// TwinCAT 3 PLC project BX130XPLC
// ProgramVersion: 3.1.4024.0
// libraries:
//   Tc2_EtherCAT, * (Beckhoff Automation GmbH)
//   Tc2_MC2, * (Beckhoff Automation GmbH)
//   Tc2_ModbusSrv, * (Beckhoff Automation GmbH)
//   Tc2_NcDrive, * (Beckhoff Automation GmbH)
//   Tc2_Standard, * (Beckhoff Automation GmbH)
//   Tc2_System, * (Beckhoff Automation GmbH)
//   Tc2_Utilities, * (Beckhoff Automation GmbH)
//   Tc3_Module, * (Beckhoff Automation GmbH)
//   TcMatrix, * (Burks Engineering)
// project tree:
//   DUTs/ E_MachineState.TcTLEO, E_ProgramMap.TcDUT, Program_Type.TcDUT, Structure_Error.TcDUT, Structure_RobotPose.TcDUT, Tool_Type.TcDUT
//   GVLs/ GVL_Axes.TcGVL, GVL_OperationCounter.TcGVL, GVL_Programs.TcGVL, GVL_SERVO_ROBOT_CONST.TcGVL
//   / PlcTask.TcTTO
//   POUs/Components/ FB_Enclosure.TcPOU, FB_GantryHoldDown.TcPOU, FB_OperatingCounter.TcPOU, FB_Robot.TcPOU, FB_Spindle.TcPOU, FB_TorqueSensor.TcPOU
//   POUs/ FB_Machine.TcPOU, MAIN.TcPOU
// real-time tasks:
//   TASK PlcTask: cycle T#10ms, priority 20, ADS port 350
// motion (NC):
//   TASK NC-Task 1 SAF: cycle T#2ms, priority 4, ADS port 501
//   TASK NC-Task 1 SVB: cycle T#10ms, priority 8, ADS port 511
//   AXIS Axis West (id 1)
//     Dynamic: Acceleration=260.052, Deceleration=260.052, Jerk=780.156
//     Velo: RefSync=10, SlowManual=8.6684051275234, FastManual=52.0104307651404, Fast=173.368102550468, Maximum=173.368
//     OtherSettings: AllowMotionCmdToSlave=true
//     encoder EncType=8
//       EncPara: ScaleFactorNumerator=9.999689, ScaleFactorDenominator=1048576, Inverse=true, MaxCount=#xffffffff
//         SoftEndMinControl: Enable=true, Range=1
//         SoftEndMaxControl: Enable=true, Range=2335
//         Inc: RefSearchInverse=true, RefSyncInverse=false
//     drive DrvType=9
//       DrvPara: Inverse=true, MaxCount=#xffffffff, DriveControlDWord=#x00030100
//         Analog: VeloReferenz=190.704912805515, VeloScale=1.02400649589962, TorqueSetpointScale=10, ScaleFactorActTorque=0.1
//         TimeComp: TaskDelayCycles=1
//     controller CtrType=1
//       CtrPara: PriorControlFactor=1
//         Observer: BandWidth=20
//   AXIS Axis East (id 2)
//     Dynamic: Acceleration=260.052, Deceleration=260.052, Jerk=780.156
//     Velo: RefSearch=1.73368102550468, RefSync=1.73368102550468, SlowManual=8.6684051275234, FastManual=52.0104307651404, Fast=173.368102550468, Maximum=173.368
//     OtherSettings: AllowMotionCmdToSlave=true
//     encoder EncType=8
//       EncPara: ScaleFactorNumerator=9.999689, ScaleFactorDenominator=1048576, MaxCount=#xffffffff
//         SoftEndMaxControl: Range=2377
//         Inc: RefSearchInverse=true, RefSyncInverse=false
//     drive DrvType=9
//       DrvPara: MaxCount=#xffffffff, DriveControlDWord=#x00030100
//         Analog: VeloReferenz=190.704912805515, VeloScale=1.02400649589962, TorqueSetpointScale=10, ScaleFactorActTorque=0.1
//         TimeComp: TaskDelayCycles=1
//     controller CtrType=1
//       CtrPara: PriorControlFactor=1
//         Observer: BandWidth=20
// I/O:
//   DEVICE PortLAN1X102, AmsNetId 172.18.239.23.3.1
//     Term 1 (EK1100) [EK1100 EtherCAT Coupler (2A E-Bus)]
//       Term 2 (EL1918) [EL1918, 8Ch. Safety Input 24V, TwinSAFE]
//         modules: Module 1 (FSOE), Module 2 (FSLOGIC)
//       Term 3 (EL1918) [EL1918, 8Ch. Safety Input 24V, TwinSAFE]
//         modules: Module 2 (FSLOGIC)
//       Term 4 (EL2904) [EL2904, 4 Ch. Safety Output 24V, 0.5A, TwinSAFE]
//         modules: Module 1 (FSOES), Module 2 (DO)
//       Term 5 (EL1008) [EL1008 8Ch. Dig. Input 24V, 3ms]
//       Term 6 (EL1008) [EL1008 8Ch. Dig. Input 24V, 3ms]
//       Term 7 (EL1008) [EL1008 8Ch. Dig. Input 24V, 3ms]
//       Term 8 (EL9410) [EL9410 E-Bus Power Supplier  (Diagnostics)]
//       Term 9 (EL2008) [EL2008 8Ch. Dig. Output 24V, 0.5A]
//       Term 10 (EL2008) [EL2008 8Ch. Dig. Output 24V, 0.5A]
//       Term 11 (EL2008) [EL2008 8Ch. Dig. Output 24V, 0.5A]
//       Term 27 (EL1008) [EL1008 8Ch. Dig. Input 24V, 3ms]
//       Term 12 (EK1122) [EK1122 2 port EtherCAT junction]
//         Term 30 (ATI Axia F/T Sensor) [ATI Axia F/T Sensor]
//       Term 15 (EL9011) [EL9011 End Terminal]
//     Drive 13 (AX5206-0000-0214) [AX5206-0000-0214 EtherCAT Drive (SoE, 2 Ch.)]
//     Box 14 (ECT I/F for KHI Robot Controller) [ECT I/F for KHI Robot Controller]
// variable links:
//   PortLAN1X102 <-> PortLAN1X102/Term 1 (EK1100)/Term 3 (EL1918)
//     Term 1 (EK1100)/Term 2 (EL1918)/Module 1 (FSOE)/FSoE Inputs/FSOE <-> ConnectionOutputs/Message_3 RxPDO
//     Term 1 (EK1100)/Term 2 (EL1918)/Module 1 (FSOE)/FSoE Outputs/FSOE <-> ConnectionInputs/Message_3 TxPDO
//     Term 1 (EK1100)/Term 4 (EL2904)/Module 1 (FSOES)/TxPDO/FSOE <-> ConnectionOutputs/Message_4 RxPDO
//   PortLAN1X102 <-> PortLAN1X102/Term 1 (EK1100)/Term 4 (EL2904)
//     Term 1 (EK1100)/Term 3 (EL1918)/ConnectionInputs/Message_4 TxPDO <-> Module 1 (FSOES)/RxPDO/FSOE
//   NC-Task 1 SAF/Axes/Axis East <-> PortLAN1X102/Drive 13 (AX5206-0000-0214)
//     Drive/Inputs/In/nDataIn1 <-> AT 2/Following distance
//     Drive/Inputs/In/nDataIn3[0] <-> AT 2/Torque/force feedback value
//     Drive/Inputs/In/nDcOutputTime <-> InfoData/DcOutputShift
//     Drive/Inputs/In/nState1 <-> AT 2/Drive status word @bit 8
//     Drive/Inputs/In/nState2 <-> AT 2/Drive status word
//     Drive/Inputs/In/nState4 @bit 1 <-> WcState/InputToggle
//     Drive/Inputs/In/nState4 <-> WcState/WcState
//     Drive/Outputs/Out/nCtrl1 <-> MDT 2/Master control word @bit 8
//     Drive/Outputs/Out/nDataOut1 <-> MDT 2/Position command value
//     Enc/Inputs/In/nDataIn1 <-> AT 2/Position feedback 1 value (motor feedback)
//     Enc/Inputs/In/nDcInputTime <-> InfoData/DcInputShift
//     Enc/Inputs/In/nState4 @bit 1 <-> WcState/InputToggle
//     Enc/Inputs/In/nState4 <-> WcState/WcState
//   NC-Task 1 SAF/Axes/Axis West <-> PortLAN1X102/Drive 13 (AX5206-0000-0214)
//     Drive/Inputs/In/nDataIn1 <-> AT 1/Following distance
//     Drive/Inputs/In/nDataIn3[0] <-> AT 1/Torque/force feedback value
//     Drive/Inputs/In/nDcOutputTime <-> InfoData/DcOutputShift
//     Drive/Inputs/In/nState1 <-> AT 1/Drive status word @bit 8
//     Drive/Inputs/In/nState2 <-> AT 1/Drive status word
//     Drive/Inputs/In/nState4 @bit 1 <-> WcState/InputToggle
//     Drive/Inputs/In/nState4 <-> WcState/WcState
//     Drive/Outputs/Out/nCtrl1 <-> MDT 1/Master control word @bit 8
//     Drive/Outputs/Out/nDataOut1 <-> MDT 1/Position command value
//     Enc/Inputs/In/nDataIn1 <-> AT 1/Position feedback 1 value (motor feedback)
//     Enc/Inputs/In/nDcInputTime <-> InfoData/DcInputShift
//     Enc/Inputs/In/nState4 @bit 1 <-> WcState/InputToggle
//     Enc/Inputs/In/nState4 <-> WcState/WcState
//   BX130XPLC/BX130XPLC Instance <-> PortLAN1X102/Box 14 (ECT I/F for KHI Robot Controller)
//     PlcTask Inputs/MAIN.fbMachine.fbRobot.jt1_pose_1 <-> TxPDO/1-8
//     PlcTask Inputs/MAIN.fbMachine.fbRobot.jt1_pose_2 <-> TxPDO/9-16
//     PlcTask Inputs/MAIN.fbMachine.fbRobot.jt2_pose_1 <-> TxPDO/17-24
//     PlcTask Inputs/MAIN.fbMachine.fbRobot.jt2_pose_2 <-> TxPDO/25-32
//     PlcTask Inputs/MAIN.fbMachine.fbRobot.jt3_pose_1 <-> TxPDO/33-40
//     PlcTask Inputs/MAIN.fbMachine.fbRobot.jt3_pose_2 <-> TxPDO/41-48
//     PlcTask Inputs/MAIN.fbMachine.fbRobot.jt4_pose_1 <-> TxPDO/49-56
//     PlcTask Inputs/MAIN.fbMachine.fbRobot.jt4_pose_2 <-> TxPDO/57-64
//     PlcTask Inputs/MAIN.fbMachine.fbRobot.jt5_pose_1 <-> TxPDO/65-72
//     PlcTask Inputs/MAIN.fbMachine.fbRobot.jt5_pose_2 <-> TxPDO/73-80
//     PlcTask Inputs/MAIN.fbMachine.fbRobot.jt6_pose_1 <-> TxPDO/81-88
//     PlcTask Inputs/MAIN.fbMachine.fbRobot.jt6_pose_2 <-> TxPDO/89-96
//     PlcTask Inputs/MAIN.fbMachine.fbRobot.sigs105112 <-> TxPDO/105-112
//     PlcTask Inputs/MAIN.fbMachine.fbRobot.sigs113120 <-> TxPDO/113-120
//     PlcTask Inputs/MAIN.fbMachine.fbRobot.sigs145152 <-> TxPDO/145-152
//     PlcTask Inputs/MAIN.fbMachine.fbRobot.sigs153160 <-> TxPDO/153-160
//     PlcTask Inputs/MAIN.fbMachine.fbRobot.sigs161168 <-> TxPDO/161-168
//     PlcTask Inputs/MAIN.fbMachine.fbRobot.sigs169176 <-> TxPDO/169-176
//     PlcTask Inputs/MAIN.fbMachine.fbRobot.sigs177184 <-> TxPDO/177-184
//     PlcTask Inputs/MAIN.fbMachine.fbRobot.sigs97104 <-> TxPDO/97-104
//     PlcTask Inputs/MAIN.fbMachine.fbRobot.ztool_pose_1 <-> TxPDO/129-136
//     PlcTask Inputs/MAIN.fbMachine.fbRobot.ztool_pose_2 <-> TxPDO/137-144
//     PlcTask Outputs/MAIN.fbMachine.fbRobot.sigs{10011008..10411048 step 80008} <-> RxPDO/{1001..1041 step 8}-{1008..1048 step 8}  (6 links)
//   BX130XPLC/BX130XPLC Instance <-> PortLAN1X102/Term 1 (EK1100)/Term 10 (EL2008)
//     PlcTask Outputs/MAIN.fbMachine.fbEnclosure.enableRollingDoor <-> Channel 3/enableRollingDoor
//     PlcTask Outputs/MAIN.fbMachine.fbEnclosure.openCloseDoor <-> Channel 4/OpenCloseDoor
//     PlcTask Outputs/MAIN.fbMachine.fbGantry.cylindersCentreSouth <-> Channel 1/SV9WorkHoldDownSouthCentre
//     PlcTask Outputs/MAIN.fbMachine.fbRobot.outRobotControlPowerOn <-> Channel 2/RobotX91ControlPowerON
//   BX130XPLC/BX130XPLC Instance <-> PortLAN1X102/Term 1 (EK1100)/Term 11 (EL2008)
//     PlcTask Outputs/MAIN.fbMachine.fbGantry.cylindersSouth <-> Channel 1/SV10WorkHoldDownSouth
//   BX130XPLC/BX130XPLC Instance <-> PortLAN1X102/Term 1 (EK1100)/Term 12 (EK1122)/Term 30 (ATI Axia F/T Sensor)
//     PlcTask Inputs/MAIN.fbMachine.fbTorqueSensor.FxCounts <-> Reading Data/FxGage0
//     PlcTask Inputs/MAIN.fbMachine.fbTorqueSensor.FyCounts <-> Reading Data/FyGage1
//     PlcTask Inputs/MAIN.fbMachine.fbTorqueSensor.FzCounts <-> Reading Data/FzGage2
//     PlcTask Inputs/MAIN.fbMachine.fbTorqueSensor.TxCounts <-> Reading Data/TxGage3
//     PlcTask Inputs/MAIN.fbMachine.fbTorqueSensor.TyCounts <-> Reading Data/TyGage4
//     PlcTask Inputs/MAIN.fbMachine.fbTorqueSensor.TzCounts <-> Reading Data/TzGage5
//   BX130XPLC/BX130XPLC Instance <-> PortLAN1X102/Term 1 (EK1100)/Term 3 (EL1918)
//     PlcTask Inputs/MAIN.fbMachine.safetyPLCComErr <-> StandardInputs/Standard Out Var 11
//     PlcTask Inputs/MAIN.fbMachine.safetyPLCEStopBlockRun <-> StandardInputs/Standard Out Var 13
//     PlcTask Inputs/MAIN.fbMachine.safetyPLCEStopOut <-> StandardInputs/Standard Out Var 9
//     PlcTask Inputs/MAIN.fbMachine.safetyPLCError <-> StandardInputs/Standard Out Var 8
//     PlcTask Inputs/MAIN.fbMachine.safetyPLCFBErr <-> StandardInputs/Standard Out Var 10
//     PlcTask Inputs/MAIN.fbMachine.safetyPLCOtherErr <-> StandardInputs/Standard Out Var 12
//     PlcTask Outputs/MAIN.fbMachine.ErrorAcknowledge <-> StandardOutputs/Standard In Var 1
//     PlcTask Outputs/MAIN.fbMachine.SafetyPLCRun <-> StandardOutputs/Standard In Var 2
//     PlcTask Outputs/MAIN.fbMachine.errorReset <-> StandardOutputs/Standard In Var 6
//   BX130XPLC/BX130XPLC Instance <-> PortLAN1X102/Term 1 (EK1100)/Term 5 (EL1008)
//     PlcTask Inputs/MAIN.fbMachine.fbEnclosure.doorIsClosed <-> Channel 4/rollingDoorClosed
//     PlcTask Inputs/MAIN.fbMachine.fbGantry.pressureSwitchHoldDown <-> Channel 2/PressureSwitch2HoldDown
//     PlcTask Inputs/MAIN.fbMachine.fbGantry.pressureSwitchSpindle <-> Channel 1/PressureSwitch1Spindle
//     PlcTask Inputs/MAIN.fbMachine.fbGantry.pressureSwitchTableClamps <-> Channel 3/PressureSwitch3TableClamps
//     PlcTask Inputs/MAIN.fbMachine.fbSpindle.pbToolChange <-> Channel 8/SpindleToolChange
//     PlcTask Inputs/MAIN.fbMachine.fbSpindle.spindleToolLocked <-> Channel 7/SpindleToolLocked
//     PlcTask Inputs/MAIN.fbMachine.fbSpindle.spindleToolOpen <-> Channel 6/SpindleToolOpen
//   BX130XPLC/BX130XPLC Instance <-> PortLAN1X102/Term 1 (EK1100)/Term 6 (EL1008)
//     PlcTask Inputs/MAIN.fbMachine.fbEnclosure.pbTableEast <-> Channel 3/TablePBEast
//     PlcTask Inputs/MAIN.fbMachine.fbEnclosure.pbTableWest <-> Channel 4/TablePBWest
//     PlcTask Inputs/MAIN.fbMachine.fbGantry.ls1NE <-> Channel 1/LimitSwitchEast
//     PlcTask Inputs/MAIN.fbMachine.fbGantry.ls3NW <-> Channel 2/LimitSwitchWest
//     PlcTask Inputs/MAIN.fbMachine.fbSpindle.tool{0..3} <-> Channel {5..8}/Tool{0..3}Present  (4 links)
//   BX130XPLC/BX130XPLC Instance <-> PortLAN1X102/Term 1 (EK1100)/Term 7 (EL1008)
//     PlcTask Inputs/MAIN.fbMachine.fbSpindle.tool{4..7} <-> Channel {1..4}/Tool{4..7}  (4 links)
//     PlcTask Inputs/MAIN.fbMachine.sHMIDustCollectionOn <-> Channel 7/FlowSensorOn
//   BX130XPLC/BX130XPLC Instance <-> PortLAN1X102/Term 1 (EK1100)/Term 9 (EL2008)
//     PlcTask Outputs/MAIN.fbMachine.fbEnclosure.cylinderTableEast <-> Channel 6/SV6TableClampEast
//     PlcTask Outputs/MAIN.fbMachine.fbEnclosure.cylinderTableWest <-> Channel 5/SV5TableClampWest
//     PlcTask Outputs/MAIN.fbMachine.fbGantry.cylindersCentreNorth <-> Channel 8/SV8WorkHoldDownNorthCentre
//     PlcTask Outputs/MAIN.fbMachine.fbGantry.cylindersNorth <-> Channel 7/SV7WorkHoldDownNorth
//     PlcTask Outputs/MAIN.fbMachine.fbSpindle.cylinderToolRelease1 <-> Channel 1/SV1ToolChange1
//     PlcTask Outputs/MAIN.fbMachine.fbSpindle.cylinderToolRelease2 <-> Channel 2/SV2ToolChange2
//     PlcTask Outputs/MAIN.fbMachine.fbSpindle.dustHoodCylinder <-> Channel 3/SV3DustBootLower
//     PlcTask Outputs/MAIN.fbMachine.fbSpindle.spindleClean <-> Channel 4/SV4SpindleClean
//   BX130XPLC/BX130XPLC Instance <-> NC-Task 1 SAF/Axes/Axis East
//     PlcTask Inputs/GVL_Axes.AxisEast.NcToPlc <-> Outputs/ToPlc
//     PlcTask Outputs/GVL_Axes.AxisEast.PlcToNc <-> Inputs/FromPlc
//   BX130XPLC/BX130XPLC Instance <-> NC-Task 1 SAF/Axes/Axis West
//     PlcTask Inputs/GVL_Axes.AxisWest.NcToPlc <-> Outputs/ToPlc
//     PlcTask Outputs/GVL_Axes.AxisWest.PlcToNc <-> Inputs/FromPlc

CONFIGURATION BX130XPLC
    RESOURCE PLC ON TwinCAT3
        TASK PlcTask(INTERVAL := T#10ms, PRIORITY := 20);
        PROGRAM MAIN WITH PlcTask : MAIN;
    END_RESOURCE
END_CONFIGURATION

// ---- DUTs/E_MachineState.TcTLEO
{attribute 'qualified_only'}
{attribute 'strict'}
{attribute 'to_string'}
TYPE E_MachineState :
(
	INITIALIZATION	:= 0,
	RUN 			:= 1,
	HOLD 			:= 2,
	ERROR	 		:= 3,
	RESET			:= 4,
	TOOLCALIBRATION := 5,
	TOOLCHANGERUN	:= 6,
	TOOLCHANGEINIT 	:= 7,
	RUNMANUAL		:= 8
);
END_TYPE

// ---- DUTs/E_ProgramMap.TcDUT
{attribute 'qualified_only'}
{attribute 'strict'}
TYPE E_ProgramMap :
(
	FrontWall := 1,
	BackWall := 2,
	Option3 := 3,
	Option4 := 4,
	Option5 := 5,
	Option6 := 6,
	Option7 := 7,
	Option8 := 8,
	Option9 := 9,
	Option10 := 10
);
END_TYPE

// ---- DUTs/Program_Type.TcDUT
TYPE Program_Type :
STRUCT
	index 				: INT;
	option1true			: STRING;
	option1false		: STRING;
	option2true			: STRING;
	option2false		: STRING;
	option3true			: STRING;
	option3false		: STRING;
	option4true			: STRING;
	option4false		: STRING;
	option5true			: STRING;
	option5false		: STRING;
	programName			: STRING;
	firstTool			: Tool_Type;
END_STRUCT
END_TYPE

// ---- DUTs/Structure_Error.TcDUT
TYPE Structure_Error :
STRUCT
	isError : BOOL := FALSE;
	errorMessage : STRING(300);
	errorType	: USINT;
END_STRUCT
END_TYPE

// ---- DUTs/Structure_RobotPose.TcDUT
TYPE Structure_RobotPose :
STRUCT
	xPose : LREAL;
	yPose : LREAL;
	zPose : LREAL;
	yPoseDustBootNorth : LREAL;
	yPoseDustBootSouth : LREAL;
	oPose : INT;
	aPose : INT;
	tPose : INT;
END_STRUCT
END_TYPE

// ---- DUTs/Tool_Type.TcDUT
TYPE Tool_Type :
STRUCT
	speed 				: INT;
	toolNumber 			: INT;
	modelName			: STRING;
	name				: STRING;
	x_coord				: INT;
	y_coord				: INT;
	z_coord				: INT;
END_STRUCT
END_TYPE

// ---- GVLs/GVL_Axes.TcGVL
{attribute 'qualified_only'}
VAR_GLOBAL
	AxisWest : AXIS_REF; // Left when facing robot
	AxisEast : AXIS_REF; // Right when facing robot
END_VAR

// ---- GVLs/GVL_OperationCounter.TcGVL
{attribute 'qualified_only'}
VAR_GLOBAL PERSISTENT
	totalRunHours : LREAL := 0;
END_VAR

// ---- GVLs/GVL_Programs.TcGVL
{attribute 'qualified_only'}
VAR_GLOBAL
	// ================= Tool Types ====================================
	//TODO: change 
	quarterInchUpcut : Tool_Type := (speed := 18000, toolNumber := 2, modelname := 'Dimar', name := 'Quarter Inch Upcut', x_coord := 0, y_coord := 125, z_coord := 446);
	halfInchUpcut : Tool_Type := (speed := 22000, toolNumber := 4, modelname := 'Dimar', name := 'Half Inch Upcut', x_coord := 0, y_coord := 134, z_coord := 454);
	sawblade : Tool_Type := (speed := 10000, toolNumber := 0, modelname := 'Hunter Precision Tools', name := 'Sawblade', x_coord := 74, y_coord := 193, z_coord := 509);
	dovetail : Tool_Type := (speed := 18000, toolNumber := 5, modelname := 'Dimar', name := 'Dovetail');
	halfInchBall : Tool_Type := (speed := 18000, toolNumber := 6, modelname := 'Dimar', name := 'Half Inch Ball');
//	quarterInchBall : Tool_Type := (speed := 18000, toolNumber := 7, modelname := 'Dimar', name := 'Quarter Inch Ball');
	noTool : Tool_Type := (speed := 0, toolNumber := 8, modelname := 'Dimar', name := 'None');

	// ================= Programs ====================================
	//Update C:\Users\kris\OneDrive\Documents\Robot transfer\Robot Programs\BX130XControlCode\BX130XControlCode\BX130XPLC\POUs\FB_Machine.TcPOU
	FrontWall : Program_Type := (index := 0, option1true := 'E cut', option1false := 'No E cut', option2true := 'Glass Door', option2false := 'Wood Door', option3true := 'Lock', option3false := 'No Lock', programName := 'Front Wall', firstTool := halfInchUpcut);
	BackWall : Program_Type := (index := 1, option1true := 'STD Window', option1false := 'No Window', option2true := 'Chimney Cut', option2false := 'No Chimney', option3true := '', option3false := '', programName := 'Back Wall', firstTool := halfInchUpcut);	
	Option3 : Program_Type := (index := 2, option1true := '', option1false := '', option2true := '', option2false := '', option3true := '', option3false := '', programName := 'Option3', firstTool := quarterInchUpcut);
	Option4 : Program_Type := (index := 3, option1true := '', option1false := '', option2true := '', option2false := '', option3true := '', option3false := '', programName := 'Option4', firstTool := quarterInchUpcut);
	ToolChange : Program_Type := (index := 10, option1true := '', option1false := '', option2true := '', option2false := '', option3true := '', option3false := '', programName := 'ToolChange', firstTool := quarterInchUpcut);
END_VAR

// ---- GVLs/GVL_SERVO_ROBOT_CONST.TcGVL
{attribute 'qualified_only'}
//Position of the robot at the centre of the gantry at max and min travel of the gantry.

VAR_GLOBAL CONSTANT
	MIN_POS_ROBOT : LREAL := 961.833; // Position of robot at min travel servo
	MAX_POS_ROBOT : LREAL := 3271.799; // Position of robot at max travel servo
	MAX_POS_SERVOWEST : LREAL := 2310; // max travel of servo
 	MIN_POS_SERVOWEST : LREAL := 1; // min travel of servo
	DIFFERENCE_ROBOT : LREAL := MAX_POS_ROBOT - MIN_POS_ROBOT; //Robot distance along gantry length
	DIFFERENCE_SERVOWEST : LREAL := MAX_POS_SERVOWEST - MIN_POS_SERVOWEST; // Total Gantry length,mm
	POSITION_LIMIT_SWITCH : LREAL := 417.4; //Position of limit switch along servo gantry, mm
	FOLLOW_THRESHOLD : LREAL := 42; //mm, min distance between dust boot and rollers kRIS MOVED IT UP FROM 24MM ON JAN 5 2026 Moved from 34mm on Jan 26 2026 Kris
	ROLLERS_Z_HEIGHT : LREAL := 800; // Robot tool z height at rollers
	ROLLERS_Z_HEIGHT_RAISED : REAL := 707; // Height of the rollers when raised, relative to robot base
	ROLLERS_Z_HEIGHT_LOWERED : REAL := 635; // Height of the rollers when lowered, relative to robot base
	INNER_ROLLERS_SPACING : LREAL := 506; //Distance between the inside ot the two centre rollers, mm
	OUTER_ROLLERS_SPACING : LREAL := 977; //Distance between the inside ot the two outer rollers, mm
	LASER_SERVO_DIFFERENCE_THRESHOLD : INT := 30; //Max allowable difference between laser position readout, and servo readout
END_VAR

// ---- POUs/MAIN.TcPOU
PROGRAM MAIN
VAR
	fbMachine				: FB_Machine;
	Run AT %Q* : BOOL := TRUE;
	ErrorAcknowledge AT %Q* : BOOL;
	errorReset AT %Q* : BOOL;
	
END_VAR

fbMachine();

END_PROGRAM

// ---- POUs/FB_Machine.TcPOU
FUNCTION_BLOCK FB_Machine //Control program
VAR_INPUT
END_VAR
VAR_OUTPUT
END_VAR
VAR
	robotPose 		: Structure_RobotPose;
	// =============== Machine Modules ================================================
	fbRobot					: FB_Robot;					// Robot object
	fbSpindle				: FB_Spindle;				// Spindle Object. Includes spindle speed, tool changing control
	fbGantry				: FB_GantryHoldDown;		// Gantry hold down object. Includes servo control, pneumatic clamping control, robot following
	fbEnclosure				: FB_Enclosure;				// Enclosure control. Includes table clamping, dust collection monitoring, door control
	fbTorqueSensor			:FB_TorqueSensor;
	fbOperatingCounter		: FB_OperatingCounter;
	
// =============== Safety ================================================
	SafetyPLCRun AT %Q* : BOOL := TRUE; //Ouput to safety PLC to run. If FALSE, safetyPLC turns off and EStop occurs
	safetyPLCEStopBlockRun AT %I* : BOOL; //Status of safety PLC Estop block. If FALSE, Estop block not running
	ErrorAcknowledge AT %Q* : BOOL; // If SafetyPLC goes into error, this needs to turn on to be able to reset
	errorReset AT %Q* : BOOL; // Resets E stops. Must be triggered to enable eStop output
	safetyPLCEStopOut AT %I* : BOOL; //Status of Estop output
	//Safety PLC Errors. If any true, Safety PLC not running properly. Most likely all the devices aren't communicating
	safetyPLCError AT %I* : BOOL; 
	safetyPLCComErr AT %I* : BOOL;
	safetyPLCFBErr AT %I* : BOOL;
	safetyPLCOtherErr AT %I* : BOOL;					
	
	// =============== State machine ================================================
	eSystemState			: E_MachineState := E_MachineState.INITIALIZATION;  // Current state 
	sHMIeSystemStateString	: STRING := TO_STRING(eSystemState); //String of current state, displayed on HMI
	eRequestedState			: E_MachineState := E_MachineState.INITIALIZATION;
	resetSuccessful			: BOOL; //Must be true to reenter initilization
	timerReset				: TON; //tIMER TO SEE HOW LONG OPERATING RESET HAS BEEN ON FOR
	startTimerReset: BOOL;
	fbgetSlaveState 		: FB_EcGetSlaveState;
	fbSetSlaveState : FB_EcSetSlaveState;
	executeGetSlaveState : BOOL;
	executeSetSlaveState : BOOL;
	timerRun				: TON; //Timer for how long Run has been on
	startTimerRun			: BOOL;
	
	// =============== HMI buttons and states ========================================
	//Universal buttons
	bHMIReset				: BOOL;	// Button to reset program
	rTrigResetErrors		: R_TRIG; //Trigger linked to bHMIReset
	sHMIErrorDisplay		: STRING(300);
	fTrigInProgramRunning 		: F_TRIG; //Trigger for when robot finishes program
	rTrigInRobotToolUpdated		: R_TRIG; //Trigger for when robot updates tool number

	// initialize.content buttons
	bHMIHomeRobot			: BOOL; 
	rTrigHomeRobot			: R_TRIG; 
	bHMIHomeMotors			: BOOL; 
	rTrigHomeMotors			: R_TRIG; 
	bHMIOpenCloseDoor		: BOOL; 
	rTrigOpenCloseDoor		: R_TRIG; 
	fTrigOpenCloseDoor		: F_TRIG; 
	bHMILockTables			: BOOL; 
	rTrigLockTables			: R_TRIG; 
	fTrigUnlockTables		: F_TRIG; 
	bHMILowerRaiseRollers	: BOOL; 
	rTrigRaiseRollers		: R_TRIG; 
	fTrigLowerRollers		: F_TRIG; 
	bHMIWarmupSpindle		: BOOL; 
	rTrigWarmupSpindle		: R_TRIG; //
	fTrigStopSpindle		: F_TRIG; //
	bHMIChangeTool			: BOOL;
	rTrigChangeTool			: R_TRIG;
	fTrigStopChangeTool		: F_TRIG;
	rTrigGoToCleanupRobot: R_TRIG;
	bHMIGoToCleanupPosition : BOOL;
	bHMIEnableInitialization: BOOL;
	
	// initialize.content indicators
	sHMICurrentTool			: INT := 8;
	sHMIRequestedTool		: INT := 8;
	sHMIDoorStatus			: STRING(80);
	
	// Settings.content buttons
	bHMIMoveServosNorth : BOOL;
	fTrigMoveServosNorth : F_TRIG;
	bHMIMoveServosSouth : BOOL;
	fTrigMoveServosSouth : F_TRIG;
	bHMIMoveRobotXneg : BOOL;
	bHMIMoveRobotXplus : BOOL;
	bHMIMoveRobotYneg : BOOL;
	bHMIMoveRobotYplus : BOOL;
	bHMIMoveRobotZneg : BOOL;
	bHMIMoveRobotZplus : BOOL;
	bHMIEnableMovement : BOOL;
	rTrigEnableMovement : R_TRIG;
	
	// settings.content indicators
	sHMISettingsMessage : STRING(80);
	// selectProgram.content inputs
	programWallChoice	: USINT; // 1 for front wall, 2 for back wall, 10 for option 3-16 for additional options
	programOption1		: BOOL; //Front wall: True: E cut, False, no e cut Back wall: True: STDWindow, False, no window
	programOption2		: BOOL; //Front wall: True: glass door, False, wood door Back wall: True: Chimney cut, False, no chimney cut
	programOption3		: BOOL; //Front wall: True: Door lock, false, no lock Back wall: NA
	bHMIRunProgramScreen		: BOOL; 
	rTrigRunProgramScreen		: R_TRIG;
	//=============Programs====================
	selectedProgram : Program_Type;
	
	// run.content buttons
	bHMIStart				: BOOL; // Button to start program. Called from Run.content
	rTrigStartProgram		: R_TRIG; //
	fTrigStopProgram		: F_TRIG; //
	bHMIHold				: BOOL; // Button to hold program. Called from Run.content
	bHMILoadTool			: BOOL; // Button to activate tool load pushbutton. Called from Run.content
	rTrigLoadTool			: R_TRIG; //
	bHMIToolLoaded			: BOOL; // Button to confirm tool is loaded. Called from Run.content
	rTrigToolLoaded			: R_TRIG; //
	bActivateRollers		: BOOL; // Button to make rollers follow robot. Called from Run.content
	escapeRunScreenEnable	: BOOL := TRUE;
	HMILeaveRunScreen		: BOOL;
	rTrigHMILeaveRunScreen	: R_TRIG;
	bHMIManual				: BOOL; // Button to switch state into manual mode. TODO: make
	
	// run.content indicators
	sHMIPneumaticsOK		: BOOL; // Indicator light of pneumatic pressure, called from run.content
	sHMIRobotHomed			: BOOL; // Indicator light of robot homed, called from run.content. Todo: Change colour/text when activated
	sHMIRollersActivated	: BOOL; // Indicator light of rollers activated, called from run.content
	sHMIeStopsOff			: BOOL; // Indicator light of e stops off, called from run.content
	sHMIDustCollectionOn AT %I*	: BOOL;
	sProgramString			: STRING;
	sHMIDisplayMessage		: STRING; //Run display
	sHMIIsError				: BOOL; //
	
	// Error states
	eInitializeServos : Structure_Error;
	powerUp				: BOOL := TRUE;
	overrideErrors		: BOOL := FALSE; //FOR  DEBUGGING PURPOSES ONLY
	disableSpindle		: BOOL := FALSE; //FOR DEBUGGING PURPOSES ONLY
	toolMatchTimer : TON;
	sHMIPopup			: BOOL;
	popupMessage		: STRING(300);
	popUpAutoReset		: BOOL;
	popupRefreshTimer: TON;
END_VAR

// Call of actions
	// Init
	overrideErrors := FALSE;
	disableSpindle := FALSE;
	//HMI update
	// Update each HMI indicator
	sHMIRobotHomed := fbRobot.inRobotAtHome;
	sHMIRollersActivated := bActivateRollers AND GVL_Axes.AxisWest.Status.Homed;
	sHMIeStopsOff := NOT fbRobot.inRobotError;
	IF fbSpindle.toolSelectedAtInitialization THEN
		sHMICurrentTool := fbSpindle.currentTool.toolNumber;
	END_IF
	sHMIeSystemStateString	:= TO_STRING(eSystemState);
	IF fbEnclosure.doorIsClosed THEN
		sHMIDoorStatus := 'Open Door';
	ELSE
		sHMIDoorStatus := 'Close Door';
	END_IF
	
	// Mode and state requests
	Change_State();  // Changes state based on inputs
	State_Machine(); // Calls functions based on state
	fbgetSlaveState(sNetId := '172.18.239.23.3.1', nSlaveAddr := 1016, bExecute := executeGetSlaveState); //slave state of controller
	
	// Update robot IOs
	fbRobot();
	robotPose := fbRobot.Update_Pose();
	fbRobot.Update_Spindle_Status(spindleStopped := fbSpindle.spindleIsStopped);
	fbGantry();
	fbEnclosure();
	fbSpindle();
	fbTorqueSensor();
	fbOperatingCounter(stateString := sHMIeSystemStateString);
	
	//Safety
	ErrorAcknowledge := safetyPLCError OR safetyPLCEStopOut OR safetyPLCComErr OR safetyPLCFBErr OR safetyPLCOtherErr;
	
// HMI button triggers
	rTrigHomeRobot(CLK := bHMIHomeRobot);
	rTrigHomeMotors(CLK := bHMIHomeMotors);
	rTrigOpenCloseDoor(CLK := bHMIOpenCloseDoor);
	rTrigLockTables(CLK := bHMILockTables);
	rTrigRaiseRollers(CLK := bHMILowerRaiseRollers);
	rTrigWarmupSpindle(CLK := bHMIWarmupSpindle);
	rTrigRunProgramScreen(CLK := bHMIRunProgramScreen);
	rTrigStartProgram(CLK := bHMIStart);
	rTrigLoadTool(CLK := bHMILoadTool);
	rTrigToolLoaded(CLK := bHMIToolLoaded);
	rTrigResetErrors(CLK := bHMIReset);
	rTrigChangeTool(CLK := bHMIChangeTool);
	rTrigGoToCleanupRobot(CLK := bHMIGoToCleanupPosition);
	rTrigEnableMovement(CLK := bHMIEnableMovement);
	
	fTrigOpenCloseDoor(CLK := bHMIOpenCloseDoor);
	fTrigUnlockTables(CLK := bHMILockTables);
	fTrigLowerRollers(CLK := bHMILowerRaiseRollers);
	fTrigStopSpindle(CLK := bHMIWarmupSpindle);
	fTrigInProgramRunning(CLK := fbRobot.inRobotProgramRunning);
	rTrigInRobotToolUpdated(CLK := fbRobot.inRobotToolUpdated);
	fTrigStopProgram(CLK := bHMIStart);
	fTrigStopChangeTool(CLK := bHMIChangeTool);
	rTrigHMILeaveRunScreen(CLK := HMILeaveRunScreen);
	fTrigMoveServosNorth(CLK := bHMIMoveServosNorth);
	fTrigMoveServosSouth(CLK := bHMIMoveServosSouth);
	
	timerReset(IN := startTimerReset, PT := t#10s);

	IF rTrigHMILeaveRunScreen.Q THEN
		fbRobot.Stop_Robot_Program(forgetProgram := TRUE);
		bHMIStart := FALSE;
		HMILeaveRunScreen := FALSE;
	ELSE
		HMILeaveRunScreen := FALSE;
	END_IF
	
	IF fbRobot.timerOutRobotStartProgram.Q THEN
		Popup_Error('Robot not started after 20 seconds. Check if robot is in cycle mode', TRUE);
	END_IF

METHOD Change_State
VAR_INPUT
END_VAR
VAR
	errorState : Structure_Error;
	temp: BOOL;
END_VAR
// Initialize -> Run
errorState := Run_Error();
IF overrideErrors = TRUE THEN
	errorState.isError := FALSE;
END_IF

IF errorState.isError AND eSystemState <> E_MachineState.RESET AND eSystemState <> E_MachineState.ERROR THEN
	escapeRunScreenEnable := TRUE;
	eSystemState := E_MachineState.ERROR;
	Popup_Error(errorState.errorMessage, TRUE);
	fbSpindle.Dust_Hood(x_pose := 0, enable := FALSE);
	eSystemState := E_MachineState.ERROR; 
	bHMIStart := FALSE;
	startTimerRun := FALSE;
END_IF

CASE eSystemState OF
	E_MachineState.ERROR:
		escapeRunScreenEnable := TRUE;
		IF rTrigResetErrors.Q THEN
			startTimerReset := TRUE;
			eSystemState := E_MachineState.RESET;
		END_IF
		
	E_MachineState.INITIALIZATION:
		escapeRunScreenEnable := TRUE;
		IF rTrigStartProgram.Q AND NOT errorState.isError THEN
			IF fbEnclosure.cylinderTableWest AND fbEnclosure.cylinderTableEast AND fbSpindle.CurrentTool.toolNumber = fbRobot.inRobotToolNumberRequest THEN
				HMILeaveRunScreen := FALSE;
				eSystemState := E_MachineState.RUN;
				fbRobot.Program_Select(programChoice := programWallChoice, option1 := programOption1, option2 := programOption2, option3 := programOption3);
				IF NOT disableSpindle THEN
					fbSpindle.Start_Spindle(spindleSpeed := fbSpindle.currentTool.speed);
				END_IF
				fbRobot.Start_Robot();
			ELSE
				Popup_Error('Tables not locked', TRUE);
			END_IF
		END_IF
		
		IF rTrigResetErrors.Q THEN
			startTimerReset := TRUE;
			eSystemState := E_MachineState.RESET;
		END_IF
		
		IF rTrigChangeTool.Q THEN
			IF fbSpindle.Verify_Tool_Change_Request(sHMICurrentTool, sHMIRequestedTool) THEN
				eSystemState := E_MachineState.TOOLCHANGEINIT;
//				fbRobot.Stop_Robot_Program(forgetProgram := TRUE);
				fbRobot.Update_Tool(current := INT_TO_USINT(sHMICurrentTool), request := INT_TO_USINT(sHMIRequestedTool));
				IF NOT fbSpindle.Update_Current_Tool(toolNumber := sHMICurrentTool) THEN
					Popup_Error('Update Tool Failed - invalid tool number', TRUE);
				END_IF
				fbRobot.Program_Select(programChoice := 10, option1 := FALSE, option2 := FALSE, option3 := FALSE);
				fbRobot.Start_Robot();
			ELSE
				Popup_Error('Tool present in destination tool holder, or tool not present in pickup tool holder. Fix and try to change tool again. If false, check tool limit switches', TRUE);
				bHMIChangeTool := FALSE;
			END_IF
		END_IF
	
//	E_MachineState.MANUALMOVE: TODO: Implement
//		
		
	E_MachineState.RUN:
		timerRun(IN := startTimerRun, PT := T#10S);
		startTimerRun := TRUE;
		escapeRunScreenEnable := FALSE;
		IF (fTrigStopProgram.Q OR fTrigInProgramRunning.Q) AND NOT errorState.isError THEN
			eSystemState := E_MachineState.INITIALIZATION;
			fbSpindle.Dust_Hood(x_pose := 0, enable := FALSE);
			fbSpindle.Stop_Spindle();
			fbRobot.Stop_Robot_Program(forgetProgram := FALSE);
			fbGantry.Lower_Raise_Rollers(raiseRollers := TRUE);
			bHMIStart := FALSE;
			startTimerRun := FALSE;
		END_IF
		
		IF fbRobot.inRobotToolNumberRequest <> fbSpindle.currentTool.toolNumber THEN
			fbSpindle.Stop_Spindle();
			fbSpindle.Dust_Hood(x_pose := 0, enable := FALSE);
			IF fbSpindle.Verify_Tool_Change_Request(fbSpindle.currentTool.toolNumber, fbRobot.inRobotToolNumberRequest) THEN
				eSystemState := E_MachineState.TOOLCHANGERUN;
			ELSE
				Popup_Error('Tool present in destination tool holder, or tool not present in pickup tool holder. Error thrown, program restart. If false, check tool limit switches', TRUE);
				eSystemState := E_MachineState.ERROR;
			END_IF
			startTimerRun := FALSE;
			toolMatchTimer(IN := FALSE);
		END_IF
		
		//Check robot tool coordinates
		toolMatchTimer(IN := NOT fbRobot.Robot_Coords_Match_Tool(current_Tool := fbSpindle.currentTool) AND fbRobot.outRobotRunHold, PT:=T#3S);
		IF toolMatchTimer.Q THEN
			Popup_Error('Tool coordinates in robot program do not match the current tools coordinates', TRUE);
			eSystemState := E_MachineState.ERROR;
			startTimerRun := FALSE;
		END_IF
		
	E_MachineState.RESET:
		escapeRunScreenEnable := TRUE;
		IF resetSuccessful THEN
			startTimerReset := False;
			eSystemState := E_MachineState.INITIALIZATION;
			bActivateRollers := FALSE;
			resetSuccessful := FALSE;
		END_IF
		
		IF timerReset.Q THEN
			startTimerReset := FALSE;
			Popup_Error('Reset unsuccessful. Check error list', TRUE);
			eSystemState := E_MachineState.ERROR;
		END_IF
		
	E_MachineState.TOOLCHANGERUN:
		IF eRequestedState := E_MachineState.RUN THEN
			eSystemState := E_MachineState.RUN;
			fbSpindle.Manual_Tool_Change(changeToolEnable := FALSE);
			fbSpindle.Start_Spindle(spindleSpeed := fbSpindle.currentTool.speed);
		END_IF
		
		//Move to change state
		fbSpindle.Update_Requested_Tool(toolNumber := fbRobot.inRobotToolNumberRequest);
		escapeRunScreenEnable := FALSE;
		
	E_MachineState.TOOLCHANGEINIT:
		escapeRunScreenEnable := TRUE;
		IF fTrigInProgramRunning.Q THEN
			IF NOT fbSpindle.Update_Current_Tool(toolNumber := fbRobot.inRobotToolNumberCurrent) THEN
				Popup_Error('Invalid tool number', TRUE);
			END_IF;
			eSystemState := E_MachineState.INITIALIZATION;
			bHMIChangeTool := FALSE;
			fbRobot.Update_Tool(current := fbRobot.inRobotToolNumberCurrent, request := fbRobot.inRobotToolNumberCurrent);
		END_IF
		
		IF fTrigStopChangeTool.Q THEN
			fbRobot.Stop_Robot_Program(forgetProgram := FALSE);
			eSystemState := E_MachineState.INITIALIZATION;
		END_IF
END_CASE
END_METHOD

METHOD Operating_Error
VAR_INPUT
END_VAR
//Turn off spindle
fbSpindle.Stop_Spindle();
//Stop robot
fbRobot.ForceStop_Robot();
//Stop Servos
fbGantry.Stop_Servos();
fbGantry.Manual_Move_Servos(1, False);
END_METHOD

METHOD Operating_Hold
VAR_INPUT
END_VAR
END_METHOD

METHOD Operating_Initialization
VAR_INPUT
END_VAR
VAR
END_VAR
//Enables pushbutton table locking capability
fbEnclosure.Table_Clamp_Control_Pushbutton();

//Keeps the spindle off for safety, redundant
IF NOT fbSpindle.spindleWarmupOn THEN
	fbSpindle.Stop_Spindle();
END_IF

//Initializes robot on power on
IF powerUp THEN
	fbRobot.Init_Robot();
	powerUp := FALSE;
END_IF

//Home robot operation on button press
IF rTrigHomeRobot.Q THEN
	fbRobot.Home_Robot();
END_IF

//Robot moves out of the way on button press
IF rTrigGoToCleanupRobot.Q THEN
	fbRobot.Go_To_Cleanup(); //TODO: test
	fbGantry.Home_Servos(robotPose);
	bActivateRollers := FALSE;
END_IF

//Home servomotors on button press
IF rTrigHomeMotors.Q THEN
	fbGantry.Lower_Raise_Rollers(raiseRollers := TRUE); //Done, tested
	eInitializeServos := fbGantry.Home_Servos(robotPose := fbRobot.robotPose); //Done, tested
	IF eInitializeServos.isError THEN
		Popup_Error(eInitializeServos.errorMessage, TRUE);
	END_IF
END_IF

//Open/close rolling door
IF rTrigOpenCloseDoor.Q THEN
	fbEnclosure.Rolling_Door_HMI_Operation(); //Done, TODO: integrate sensor
END_IF

IF fTrigOpenCloseDoor.Q THEN
	fbEnclosure.Rolling_Door_HMI_Operation(); //Done, tested no door
END_IF

//Lock/unlock tables
IF rTrigLockTables.Q THEN
	fbEnclosure.Table_Clamp_Control_HMI(eastTableLock := TRUE, westTableLock := TRUE); //Done, tested
END_IF

IF fTrigUnlockTables.Q THEN
	fbEnclosure.Table_Clamp_Control_HMI(eastTableLock := FALSE, westTableLock := FALSE); //Done, tested
END_IF

//Raise/lower rollers
IF rTrigRaiseRollers.Q THEN
	fbGantry.Lower_Raise_Rollers(raiseRollers := TRUE); //Done, tested
END_IF

IF fTrigLowerRollers.Q THEN
	fbGantry.Lower_Raise_Rollers(raiseRollers := FALSE); //Done, tested
END_IF

//Warmup spindle
IF rTrigWarmupSpindle.Q THEN
	IF fbSpindle.toolSelectedAtInitialization AND fbSpindle.currentTool.toolNumber <> 0 THEN
		fbSpindle.Spindle_Warmup(); //Done, tested. TODO: Change spindle is warm flag if spindle hasn't been on for >3 hours
	ELSE
		Popup_Error('Tool hasnt been picked (change tool), OR sawblade loaded', TRUE);
		bHMIWarmupSpindle := FALSE;
	END_IF
END_IF

IF fbSpindle.fTrigWarm3.Q THEN
	bHMIWarmupSpindle := FALSE;
END_IF

IF fTrigStopSpindle.Q THEN
	fbSpindle.Stop_Spindle(); 
END_IF

//Save program to robot and PLC
IF rTrigRunProgramScreen.Q THEN
	fbRobot.Program_Select(programChoice := programWallChoice, option1 := programOption1, option2 := programOption2, option3 := programOption3);
	Update_Program_String();
	bHMIRunProgramScreen := FALSE;
END_IF

//Update requested tool for display on HMI
IF rTrigInRobotToolUpdated.Q THEN
	fbSpindle.Update_Requested_Tool(toolNumber := fbRobot.inRobotToolNumberRequest);
END_IF

//Manual tool change enabled if spindle is stopped
IF fbSpindle.spindleIsStopped THEN
	fbSpindle.Manual_Tool_Change(changeToolEnable := TRUE);
END_IF

//Activate Rollers
IF bActivateRollers THEN
	IF GVL_Axes.AxisWest.Status.Homed THEN
		IF fbRobot.inRobotPoseDataIsSent THEN
			fbGantry.Follow_Robot(robotPoseGantry := robotPose);
		ELSE
			Popup_Error('Robot posedata program not running', TRUE);
			bActivateRollers := FALSE;
		END_IF
	ELSE
		Popup_Error('Gantry not homed', TRUE);
		bActivateRollers := FALSE;
	END_IF
END_IF

//Jog rollers
IF bHMIMoveServosNorth THEN
	IF GVL_Axes.AxisWest.Status.Homed AND GVL_Axes.AxisEast.Status.Coupled THEN
		fbGantry.Manual_Move_Servos(direction := -1, moveServos := TRUE);
		sHMISettingsMessage := '';
	ELSE
		sHMISettingsMessage := 'Motor not homed or coupled';
	END_IF
END_IF

IF bHMIMoveServosSouth THEN
	IF GVL_Axes.AxisWest.Status.Homed AND GVL_Axes.AxisEast.Status.Coupled THEN
		fbGantry.Manual_Move_Servos(direction := 1, moveServos := TRUE);
		sHMISettingsMessage := '';
	ELSE
		sHMISettingsMessage := 'Motor not homed or coupled';
	END_IF
END_IF

IF fTrigMoveServosNorth.Q OR fTrigMoveServosSouth.Q THEN
	fbGantry.Manual_Move_Servos(direction := -1, moveServos := FALSE);
END_IF

IF rTrigEnableMovement.Q THEN
	fbRobot.Program_Select(programChoice := 11, TRUE, TRUE, TRUE);
	fbRobot.Start_Robot();
END_IF
END_METHOD

METHOD Operating_ManualMove
VAR_INPUT
END_VAR
END_METHOD

METHOD Operating_Reset
VAR_INPUT
END_VAR
VAR
	robotReset	: BOOL;
	gantryReset : BOOL;
	spindleReset : BOOL;
	state           : ST_EcSlaveState;
	count			: INT;
END_VAR
//Robot reset
robotReset := fbRobot.Reset_Robot();
//Servo Reset
gantryReset := fbGantry.Reset_Servos();
//VFD Reset
spindleReset := fbSpindle.Reset_Drive();
//Safety Reset
IF NOT safetyPLCEStopOut THEN
	errorReset := NOT errorReset;
END_IF

executeGetSlaveState := NOT executeGetSlaveState;

IF NOT fbgetSlaveState.bBusy THEN
	state := fbgetSlaveState.state;
	executeSetSlaveState := NOT executeSetSlaveState;
	//IF NOT executeGet
	CASE state.deviceState OF
		1:
			fbSetSlaveState(sNetId := '172.18.239.23.3.1', nSlaveAddr := 1016, bExecute := executeSetSlaveState, reqState := 2);
		2:
			fbSetSlaveState(sNetId := '172.18.239.23.3.1', nSlaveAddr := 1016, bExecute := executeSetSlaveState, reqState := 4);
		4:
			fbSetSlaveState(sNetId := '172.18.239.23.3.1', nSlaveAddr := 1016, bExecute := executeSetSlaveState, reqState := 8);
		8: 
		0:
		ELSE
			fbSetSlaveState(sNetId := '172.18.239.23.3.1', nSlaveAddr := 1016, bExecute := executeSetSlaveState, reqState := 1);
	END_CASE
ELSE
//	executeGetSlaveState := FALSE;
//	executeSetSlaveState := FALSE;
END_IF

IF robotReset AND gantryReset AND spindleReset AND safetyPLCEStopOut THEN
	resetSuccessful := TRUE;
	errorReset := FALSE;
END_IF
END_METHOD

METHOD Operating_Run
VAR
	robotRun : BOOL;
	toolNumber: INT;
END_VAR
// Follow robot
IF fbRobot.inRobotPoseDataIsSent THEN
	robotRun := fbGantry.Follow_Robot(robotPoseGantry := fbRobot.robotPose);
ELSE 
	robotRun := FALSE;
	Popup_Error('Robot pose data not being sent', TRUE);
END_IF

IF fbSpindle.spindleIsStopped THEN
	fbSpindle.Start_Spindle(spindleSpeed := fbSpindle.currentTool.speed);
END_IF

IF ABS(fbSpindle.spindleSpeed - fbSpindle.CurrentTool.speed) > 2000 THEN
	IF timerRun.Q THEN
		Popup_Error('Spindle not up to speed after 10s', TRUE);
	END_IF
	robotRun := FALSE;
END_IF

fbGantry.Cylinder_Set_Cutting();

//dust boot
fbSpindle.Dust_Hood(x_pose := fbRobot.robotPose.xPose, enable := TRUE);

IF bHMIHold THEN
	fbRobot.RunHold_Robot(RunHold := FALSE);
ELSE
	fbRobot.RunHold_Robot(RunHold := robotRun);
END_IF
END_METHOD

METHOD Operating_ToolChangeInit : BOOL
VAR_INPUT
END_VAR
fbSpindle.Stop_Spindle();
fbSpindle.Dust_Hood(x_pose := 0, enable := FALSE);

//Tool change auto
IF fbRobot.inRobotReleaseTool THEN
	fbSpindle.Release_Tool();
	fbRobot.Release_Update(release := fbSpindle.spindleToolOpen);
ELSE
	fbSpindle.Grab_Tool();
	fbRobot.Release_Update(release := NOT fbSpindle.spindleToolLocked);
END_IF
END_METHOD

METHOD Operating_ToolChangeRun : BOOL
VAR_INPUT
END_VAR
VAR
	runHoldToolChangeRun : BOOL := TRUE;
END_VAR
//Ensure Spindle stays off and dust hood raised
fbSpindle.Stop_Spindle();
fbSpindle.Dust_Hood(x_pose := 0, enable := FALSE);

//Release tool when requested by robot
IF fbRobot.inRobotReleaseTool THEN
	fbSpindle.Release_Tool();
	fbRobot.Release_Update(release := fbSpindle.spindleToolOpen);
ELSE
	fbSpindle.Grab_Tool();
	fbRobot.Release_Update(release := NOT fbSpindle.spindleToolLocked);
END_IF

//If robot is done tool change
IF fbRobot.inRobotToolNumberRequest = fbRobot.inRobotToolNumberCurrent THEN
	popupRefreshTimer(IN:=TRUE, PT :=T#10S); //Timer to not have constant popups
	IF popupRefreshTimer.Q THEN
		Popup_Error(CONCAT(CONCAT('Press tool loaded if ', fbSpindle.currentTool.name), ' is loaded to resume program. If not, can hold green button on spindle for three seconds to change manually'), TRUE);
		popupRefreshTimer(IN:=FALSE, PT :=T#10S);
	END_IF
	IF NOT fbSpindle.Update_Current_Tool(toolNumber := fbRobot.inRobotToolNumberCurrent) THEN
		Popup_Error('Invalid tool number', TRUE);
	END_IF;			
	runHoldToolChangeRun := FALSE;
	fbSpindle.Manual_Tool_Change(changeToolEnable := TRUE);
	IF rTrigToolLoaded.Q THEN
		eRequestedState := E_MachineState.RUN;
	END_IF
END_IF

IF (fTrigStopProgram.Q OR fTrigInProgramRunning.Q) THEN
	fbSpindle.Manual_Tool_Change(changeToolEnable := FALSE);
	eRequestedState := E_MachineState.INITIALIZATION;
	eSystemState := E_MachineState.INITIALIZATION;
	fbSpindle.Dust_Hood(x_pose := 0, enable := FALSE);
	fbSpindle.Stop_Spindle();
	fbRobot.Stop_Robot_Program(forgetProgram := FALSE);
	fbGantry.Lower_Raise_Rollers(raiseRollers := TRUE);
	bHMIStart := FALSE;
	HMILeaveRunScreen := TRUE;
	IF fbRobot.inRobotToolNumberRequest = fbRobot.inRobotToolNumberCurrent THEN
		IF NOT fbSpindle.Update_Current_Tool(toolNumber := fbRobot.inRobotToolNumberCurrent) THEN
			Popup_Error('Invalid tool number', TRUE);
		END_IF;	
	END_IF
END_IF

IF bHMIHold THEN
	fbRobot.RunHold_Robot(RunHold := FALSE);
ELSE
	fbRobot.RunHold_Robot(RunHold := runHoldToolChangeRun);
END_IF
END_METHOD

METHOD Popup_Error : BOOL
VAR_INPUT
	message : STRING (300);
	automaticReset : BOOL;
END_VAR
popupMessage := message;
sHMIpopup := TRUE;
popUpAutoReset := automaticReset;
END_METHOD

METHOD Run_Error : Structure_Error
VAR_INPUT
END_VAR
VAR
	//0: robot, 1: servos, 2: E-stops, 3: Door, 4: Pneumatics, 5: Spindle, 6: Tool changing
	pneumaticsError : Structure_Error;
END_VAR
Run_Error.errorMessage := '';
Run_Error.isError := FALSE;
//Robot Error
IF fbRobot.inRobotError THEN
	Run_Error.errorMessage := CONCAT(Run_Error.errorMessage,'\nRobot error, check teach pendant');
	Run_Error.isError := TRUE;
	Run_Error.errorType.0 := TRUE;
ELSE
	Run_Error.errorType.0 := TRUE;
END_IF

IF NOT fbRobot.inRobotPoseDataIsSent THEN
	Run_Error.isError := TRUE;
	Run_Error.errorType.0 := TRUE;
	Run_Error.errorMessage := CONCAT(Run_Error.errorMessage,'\nRobot pose data program not running');
END_IF

IF fbRobot.inRobotEStopOn THEN
	Run_Error.errorMessage := CONCAT(Run_Error.errorMessage, '\nRobot E Stop On');
	Run_Error.isError := TRUE;
	Run_Error.errorType.2 := TRUE;
ELSE
	Run_Error.errorType.2 := FALSE;
END_IF


//Servos error
IF GVL_Axes.AxisWest.Status.Error THEN
	Run_Error.errorMessage := CONCAT(Run_Error.errorMessage, CONCAT('\nwest gantry error: ', UDINT_TO_STRING(GVL_Axes.AxisWest.Status.ErrorID)));
	Run_Error.isError := TRUE;
	Run_Error.errorType.1 := TRUE;
ELSE
	Run_Error.errorType.1 := FALSE;
END_IF

IF GVL_Axes.AxisEast.Status.Error THEN
	Run_Error.errorMessage := CONCAT(Run_Error.errorMessage, CONCAT('\neast gantry error: ', UDINT_TO_STRING(GVL_Axes.AxisWest.Status.ErrorID)));
	Run_Error.isError := TRUE;
	Run_Error.errorType.1 := TRUE;
ELSE
	Run_Error.errorType.1 := FALSE;
END_IF

//Torque sensor error Todo: implement

//E-stop/safety system error Todo: 
IF NOT safetyPLCEStopOut THEN
	Run_Error.isError := TRUE;
	Run_Error.errorType.2 := TRUE;
	Run_Error.errorMessage := CONCAT(Run_Error.errorMessage, '\nSafety PLC in Error');
END_IF

//Door error
//IF fbEnclosure.doorIsOpen THEN
//	Run_Error.errorMessage := CONCAT(Run_Error.errorMessage,'\nDoorIsOpen');
//	Run_Error.isError := TRUE;
//	Run_Error.errorType.3 := TRUE;
//ELSE
//	Run_Error.errorType.3 := FALSE;
//END_IF

//Pneumatics error
pneumaticsError := fbGantry.Pneumatics_Error();

IF pneumaticsError.isError THEN
	Run_Error.errorMessage := CONCAT(Run_Error.errorMessage, pneumaticsError.errorMessage);
	Run_Error.isError := TRUE;
	Run_Error.errorType.4 := TRUE;
	sHMIPneumaticsOK := FALSE;
ELSE
	Run_Error.errorType.4 := FALSE;
	sHMIPneumaticsOK := TRUE;
END_IF

//Spindle error
IF fbSpindle.spindleError THEN
	Run_Error.errorMessage := CONCAT(Run_Error.errorMessage, '\nSpindleError');
	Run_Error.isError := TRUE;
	Run_Error.errorType.5 := TRUE;
ELSE 
	Run_Error.errorType.5 := FALSE;
END_IF

sHMIIsError := Run_Error.isError;
IF Run_Error.errorMessage = '' THEN
	sHMIErrorDisplay := 'No Errors';
ELSE
	sHMIErrorDisplay := MID(Run_Error.errorMessage, LEN(Run_Error.errorMessage) - 1, 3);
END_IF
END_METHOD

// Calls functions based on state
METHOD State_Machine 
VAR_INPUT
END_VAR
CASE eSystemState OF
	E_MachineState.INITIALIZATION:
		Operating_Initialization();
	
//	E_MachineState.MANUALMOVE:
//		Operating_ManualMove(); //TODO: Implement
		
	E_MachineState.RUN:
		Operating_Run();
		
	E_MachineState.RESET:
		Operating_Reset();
		
	E_MachineState.ERROR:
		Operating_Error();
		
	E_MachineState.TOOLCHANGERUN:
		Operating_ToolChangeRun();
		
	E_MachineState.TOOLCHANGEINIT:
		Operating_ToolChangeInit();
END_CASE
END_METHOD

METHOD Update_Program_String
VAR
	option1string			: STRING;
	option2string			: STRING;
	option3string			: STRING;
END_VAR
CASE programWallChoice OF
        1: selectedProgram := GVL_Programs.FrontWall;
        2: selectedProgram := GVL_Programs.BackWall;
        3: selectedProgram := GVL_Programs.Option3;
        4: selectedProgram := GVL_Programs.Option4;
        // Add more cases for additional options if needed
        ELSE
            // Handle invalid program wall choice
    END_CASE;

IF programOption1 THEN
	option1string := selectedProgram.option1true;
ELSE
	option1string := selectedProgram.option1false;
END_IF

IF programOption2 THEN
	option2string := selectedProgram.option2true;
ELSE
	option2string := selectedProgram.option2false;
END_IF

IF programOption3 THEN
	option3string := selectedProgram.option3true;
ELSE
	option3string := selectedProgram.option3false;
END_IF

sProgramString := CONCAT(CONCAT(CONCAT(CONCAT(CONCAT(CONCAT(selectedProgram.programName,' - '), option1string),' - '),option2string),' - '), option3string);
END_METHOD

END_FUNCTION_BLOCK

// ---- POUs/Components/FB_Robot.TcPOU
//Todo - Add flags for if communicating, program info, 
FUNCTION_BLOCK FB_Robot
VAR_INPUT
END_VAR
VAR_OUTPUT
END_VAR
VAR
	robotPose 		: Structure_RobotPose;	//Stores robot pose

	//----------Inputs From Robot ----------
	jt1_pose_1 AT %I* 		: USINT; //Signal 1-8
	jt1_pose_2 AT %I* 		: USINT; //Signal 9-16
	jt2_pose_1 AT %I* 		: USINT; //Signal 17-25
	jt2_pose_2 AT %I* 		: USINT; //Signal 26-32
	jt3_pose_1 AT %I* 		: USINT; //Signal 33-40
	jt3_pose_2 AT %I* 		: USINT; //Signal 41-48
	jt4_pose_1 AT %I* 		: USINT; //Signal 49-56
	jt4_pose_2 AT %I* 		: USINT; //Signal 57-64
	jt5_pose_1 AT %I* 		: USINT; //Signal 65-72
	jt5_pose_2 AT %I* 		: USINT; //Signal 73-80
	jt6_pose_1 AT %I* 		: USINT; //Signal 81-88
	jt6_pose_2 AT %I* 		: USINT; //Signal 89-96
	inRobotMotorOn			: BOOL; //Signal number 97
	inRobotError			: BOOL; //Signal 98
	inRobotAutomaticMode	: BOOL; //Signal 99
	inRobotAtHome			: BOOL; //Signal 100
	inRobotInTeach			: BOOL; //Signal 101
	inRobotCycleStart		: BOOL; //Signal 102
	inRobotPowerOn			: BOOL; //Signal 103
	inRobotPoseDataIsSent	: BOOL; //Signal 104
	inRobotEStopOn			: BOOL; //Signal 105
	inRobotBatteryAlarm		: BOOL; //Signal 106
	inRobotToolNumberCurrent: USINT; //Signal 107-110
	inRobotToolNumberRequest: USINT; //Signal 111-114
	inRobotReleaseTool		: BOOL; //Signal 115
	inRobotProgramRunning	: BOOL; //Signal 116
	inRobotToolUpdated		: BOOL; //Signal 117
	inRobotStartofProgram	: BOOL; //Signal 118
	sigs97104 AT %I*		: USINT;
	sigs105112 AT %I*		: USINT;
	sigs113120 AT %I*		: USINT;
	ztool_pose_1 AT %I* 	: USINT; //Signal 129-136
	ztool_pose_2 AT %I* 	: USINT; //Signal 137-144
	sigs145152 AT %I*		: USINT;
	sigs153160 AT %I*		: USINT;
	sigs161168 AT %I*		: USINT;
	sigs169176 AT %I*		: USINT;
	sigs177184 AT %I*		: USINT;
	tool_coords_x 			: USINT; //Signal 145-156
	tool_coords_y 			: USINT; //Signal 157-168
	tool_coords_z 			: USINT; //Signal 169-180
	currentTool				: Tool_Type;
	
	
	//----------Outputs To Robot ----------
	outRobotControlPowerOn AT %Q*	: BOOL := TRUE;
	outRobotTurnMotorOn				: BOOL; //Signal 1001
	outRobotResetError				: BOOL; //Signal 1002
	outRobotStartCycle				: BOOL; //Signal 1003
	outRobotResetProgram			: BOOL; //Signal 1004
	outRobotStartProgram			: BOOL; //Signal 1005
	outRobotRunHold		 			: BOOL; //Signal 1006
	outRobotHome					: BOOL; //Signal 1007
	outRobotTurnMotorOff			: BOOL; //1008
	outRobotToolReleased			: BOOL; //Signal 1009
	outRobotCurrentTool				: USINT; //Signal 1010-1013
	outRobotNoEStop					: BOOL := TRUE; //Signal 1014
	outRobotSpindleStopped			: BOOL; //Signal 1016
	outRobotProgramChoice			: USINT; //Signals 1017-1020
	outRobotProgramOption1			: BOOL; //Signal 1021
	outRobotProgramOption2			: BOOL; //Signal 1022
	outRobotProgramOption3			: BOOL; //Signal 1023
	outRobotRequestedTool			: USINT; //Signal 1024-1027
	outRobotProgramSelected			: BOOL; //Signal 1028
	outRobotGoToCleanupPosition		: BOOL; // Signal 1029 
	outRobotMoveX					: BOOL; // Signal 1030
	outRobotMoveY					: BOOL; // Signal 1031
	outRobotMoveZ					: BOOL; // Signal 1032
	outRobotMovePositive			: BOOL; // Signal 1033
	
	sigs10011008	AT %Q*			: USINT;
	sigs10091016	AT %Q*			: USINT;
	sigs10171024	AT %Q*			: USINT;
	sigs10251032	AT %Q*			: USINT;
	sigs10331040	AT %Q*			: USINT;
	sigs10411048	AT %Q*			: USINT;
	timerOutRobotStartProgram		: TON;
	
END_VAR

Update_Status();

	IF outRobotResetProgram AND inRobotStartofProgram THEN
		outRobotStartCycle := TRUE;
		outRobotResetProgram := FALSE;
	END_IF
	
	IF inRobotCycleStart AND NOT inRobotStartofProgram THEN
		outRobotStartCycle := FALSE;
	END_IF
	
	IF NOT inRobotCycleStart AND inRobotStartofProgram THEN
		outRobotStartCycle := NOT outRobotStartCycle;
	END_IF
	
	//Turn off startRobot once program started TODO: Turn off after 5 seconds
	IF inRobotProgramRunning THEN
		outRobotStartProgram := FALSE;
		outRobotGoToCleanupPosition := FALSE;
	END_IF

//Change request to home robot once robot is in home position
	IF inRobotAtHome OR inRobotError THEN 
		outRobotHome := FALSE;
	END_IF
	
//Turn off error reset and motor when on
	IF NOT inRobotError THEN
		outRobotResetError := FALSE;
	END_IF
	
	IF inRobotMotorOn THEN		
		outRobotTurnMotorOn := TRUE;
	END_IF
	
	//Switch to main program TODO
	timerOutRobotStartProgram(IN := outRobotStartProgram, PT := T#30S);
	IF timerOutRobotStartProgram.Q THEN
		outRobotStartProgram := FALSE;
	END_IF

//Turns external Estop off
METHOD EStop_OFF : BOOL
VAR_INPUT
END_VAR
outRobotNoEStop := TRUE;
END_METHOD

//E-stop to robot
METHOD ForceStop_Robot : BOOL
VAR_INPUT
END_VAR
outRobotNoEStop := FALSE;
END_METHOD

METHOD Go_To_Cleanup : BOOL
VAR_INPUT
END_VAR
outRobotGoToCleanupPosition := TRUE;
END_METHOD

//Send home command to robot
METHOD Home_Robot
VAR_INPUT
END_VAR
outRobotHome := TRUE;
END_METHOD

METHOD Init_Robot : BOOL
VAR_INPUT
END_VAR
outRobotResetError := TRUE;
outRobotTurnMotorOn := TRUE;
outRobotRunHold := TRUE;
outRobotStartCycle := TRUE;
END_METHOD

// Select the robot program based on HMI inputs
METHOD Program_Select
VAR_INPUT
	programChoice :	USINT;
	option1 : BOOL;
	option2 : BOOL;
	option3 : BOOL;
END_VAR
outRobotProgramChoice := programChoice;
outRobotProgramOption1 := option1;
outRobotProgramOption2	:= option2;
outRobotProgramOption3	:= option3;
outRobotProgramSelected := TRUE;
END_METHOD

METHOD Release_Update
VAR_INPUT
	release : BOOL;
END_VAR
outRobotToolReleased := release;
END_METHOD

//Resets robot errors
METHOD Reset_Robot : BOOL //Returns true if robot reset successfully
VAR_INPUT
END_VAR
outRobotNoEStop := TRUE;
outRobotResetError := TRUE;
outRobotTurnMotorOn := TRUE;
outRobotTurnMotorOff := FALSE;
outRobotRunHold := TRUE;
outRobotStartProgram := FALSE;
Reset_Robot := NOT(inRobotError OR inRobotEStopOn);
IF Reset_Robot THEN
	Stop_Robot_Program(forgetProgram := FALSE);
END_IF
END_METHOD

METHOD Robot_Coords_Match_Tool : BOOL
VAR_INPUT
	current_Tool : TOOL_TYPE;
END_VAR
VAR
	tooltransform : ARRAY[1..3] OF LREAL;
	sigs145160 : UINT := sigs153160*256 + sigs145152;
	sigs153168 : UINT := sigs161168*256 + sigs153160;
	sigs169184 : UINT := sigs177184*256 + sigs169176;
END_VAR
tooltransform[1] := (sigs145160 AND 16#FFF) - 4094/2; //Bits 145-156, x value
tooltransform[2] := SHR((sigs153168 AND 16#FFF0), 4) - 4094/2; // Bits 157-168, y value
tooltransform[3] := (sigs169184 AND 16#FFF) - 4094/2; // Bits 169-180, z value

IF ABS(current_Tool.x_coord - tooltransform[1]) < 2 AND ABS(current_Tool.y_coord - tooltransform[2]) < 2 AND ABS(current_Tool.z_coord - tooltransform[3]) < 2 THEN
	Robot_Coords_Match_Tool := TRUE;
ELSE
	Robot_Coords_Match_Tool := FALSE;
END_IF
END_METHOD

//TODO: Implement
METHOD Robot_Manual_Control
VAR_INPUT
END_VAR
END_METHOD

//Holds robot if false
METHOD RunHold_Robot
VAR_INPUT
	RunHold : BOOL; //True for run, False for hold
END_VAR
outRobotRunHold := RunHold;
END_METHOD

//STart robot program
METHOD Start_Robot
VAR_INPUT
END_VAR
outRobotTurnMotorOn := TRUE;
outRobotStartProgram := TRUE;
END_METHOD

METHOD Stop_Robot_Program : BOOL
VAR_INPUT
	forgetProgram : BOOL;
END_VAR
outRobotResetProgram := TRUE;
IF forgetProgram THEN
	outRobotProgramSelected := FALSE;
END_IF
RunHold_Robot(RunHold := True);
END_METHOD

//Updates current robot pose
//TODO make flag that verifies pose is being sent
METHOD Update_Pose : Structure_RobotPose
VAR_INPUT
END_VAR
VAR
	dustBoot : Array2DStaticMatrix; //This instance is the matrix that the code will interact with
	dustBoot_Data : ARRAY[1..4,1..1] OF LREAL := [-58.997,133.95,455.3,1]; //centre coordinates wrt robot flange
	dustBoot_NE : ARRAY[1..4,1..1] OF LREAL := [102.900,157.511, 283,1];
	dustBoot_SE : ARRAY[1..4,1..1] OF LREAL := [104.4,-25.4,463.580,1];
	dustBoot_SW : ARRAY[1..4,1..1] OF LREAL := [-100.52,-23.366,463.9,1];
	dustBoot_NW : ARRAY[1..4,1..1] OF LREAL := [-101.4,156.4,284,1];
	dustBoot_SRightCorner : ARRAY[1..4,1..1] OF LREAL := [-211, 32, 405.187,1];
	dustBoot_NRightCorner : ARRAY[1..4,1..1] OF LREAL := [-210.197,98.825,339.353,1];
	dustBootCornersMatrix : ARRAY[1..6] OF Array2DStaticMatrix;
	dustBootCornersData : ARRAY[1..6] OF ARRAY[1..4,1..1] OF LREAL := [[102.900,157.511, 283,1], [104.4,-25.4,463.580,1], [-100.52,-23.366,463.9,1], [-101.4,156.4,284,1], [-211, 32, 405.187,1], [-210.197,98.825,339.353,1]];
	
	maxY : LREAL;
	minY : LREAL;
	
	joints : ARRAY[1..6] OF LREAL;
	jointsrad : ARRAY[1..6] OF LREAL;
	alpha : ARRAY[1..6] OF LREAL := [-PI/2,PI,PI/2,PI/2,PI/2,0];
	theta : ARRAY[1..6] OF LREAL := [PI/2,PI/2,-PI,-PI,PI,PI/2];
	d : ARRAY[1..6] OF LREAL := [530,0,0,1650,0,225];
	a : ARRAY[1..6] OF LREAL := [200,-1160,230,0,0,0];
	
	dh : ARRAY[1..6] OF Array2DStaticMatrix;
	dh_data : ARRAY[1..6] OF ARRAY[1..4,1..4] OF LREAL;
	temp : ARRAY[1..5] OF Array2DStaticMatrix;
	temp_data : ARRAY[1..5] OF ARRAY[1..4,1..4] OF LREAL;
	i : INT;
	
	Result : Array2DStaticMatrix; //This instance is the resulting column vector
	Result_Data : ARRAY[1..4,1..1] OF LREAL := [1, 2, 3,1]; //This array will act as the memory for the resulting column vector
	
	Corners : ARRAY[1..6] OF Array2DStaticMatrix; //This instance is the resulting column vector
	Corners_Data : ARRAY[1..6] OF ARRAY[1..4,1..1] OF LREAL; //This array will act as the memory for the resulting column vector
	
	success : ARRAY[1..13] OF BOOL; //records success or failure of the matrix multiplication
	equal : BOOL; //records success if the resulting vector is equal to the first
	zpose:LREAL;
END_VAR
// RobotPose
joints[1] := -((UINT_TO_LREAL(jt1_pose_2)*256 + UINT_TO_LREAL(jt1_pose_1) - 40000)/100);
joints[2] := ((UINT_TO_LREAL(jt2_pose_2)*256 + UINT_TO_LREAL(jt2_pose_1) - 40000)/100);
joints[3] := ((UINT_TO_LREAL(jt3_pose_2)*256 + UINT_TO_LREAL(jt3_pose_1) - 40000)/100);
joints[4] := ((UINT_TO_LREAL(jt4_pose_2)*256 + UINT_TO_LREAL(jt4_pose_1) - 40000)/100);
joints[5] := ((UINT_TO_LREAL(jt5_pose_2)*256 + UINT_TO_LREAL(jt5_pose_1) - 40000)/100);
joints[6] := ((UINT_TO_LREAL(jt6_pose_2)*256 + UINT_TO_LREAL(jt6_pose_1) - 40000)/100);

zpose := ((UINT_TO_LREAL(ztool_pose_2)*256 + UINT_TO_LREAL(ztool_pose_1) - 4000));

dustBoot(Data := dustBoot_Data);
Result(Data := Result_Data);
FOR i := 1 TO 6 DO
	jointsrad[i] := DEG_TO_RAD(joints[i]);
	dh[i](Data := dh_Data[i]);
	dh[i].Denavit_Hartenberg(jt := jointsrad[i], theta := theta[i], alpha := alpha[i], d := d[i], a := a[i]);
END_FOR

FOR i := 1 TO 5 DO
	temp[i](Data := temp_data[i]);
END_FOR

success[1] := Matrix_Product(dh[1], dh[2], temp[1]);

FOR i := 2 TO 5 DO
	success[i] := Matrix_Product(temp[i-1], dh[i+1], temp[i]);
END_FOR

success[7] := Matrix_Product(temp[5],dustBoot,Result);
maxY := -5000;
minY := 5000;
FOR i := 1 TO 6 DO
	Corners[i](Data := Corners_Data[i]);
	dustBootCornersMatrix[i](Data := dustBootCornersdata[i]);
	success[i+7] := Matrix_Product(temp[5],dustBootCornersMatrix[i],corners[i]);
	IF corners[i].GetI(1) > maxY THEN
		maxY := corners[i].GetI(1);
	END_IF
	IF corners[i].GetI(1) < minY THEN
		minY := corners[i].GetI(1);
	END_IF
END_FOR

robotPose.xPose := Result.GetI(0);
robotPose.yPose := (maxY + minY) / 2;
robotPose.zPose := zpose;
Update_Pose := robotPose;
END_METHOD

METHOD Update_Spindle_Status : BOOL
VAR_INPUT
	spindleStopped : BOOL;
END_VAR
outRobotSpindleStopped := spindleStopped;
END_METHOD

//Updates run status and IOs in Beckhoff system
METHOD Update_Status
VAR_INPUT
END_VAR
// Robot signals
sigs10011008.0 := outRobotTurnMotorOn; // 1001
sigs10011008.1 := outRobotResetError; //1002
sigs10011008.2 := outRobotStartCycle; //1003
sigs10011008.3 := outRobotResetProgram; //1004
sigs10011008.4 := outRobotStartProgram; //1005
sigs10011008.5 := outRobotRunHold; //1006
sigs10011008.6 := outRobotHome; //1007
sigs10011008.7 := outRobotTurnMotorOff; //1008
sigs10091016.0 := outRobotToolReleased; //1009
sigs10091016.1 := outRobotCurrentTool.0; //1010
sigs10091016.2 := outRobotCurrentTool.1; //1011
sigs10091016.3 := outRobotCurrentTool.2; //1012
sigs10091016.4 := outRobotCurrentTool.3; //1013
sigs10091016.5 := outRobotNoEStop; //1014
sigs10091016.7 := outRobotSpindleStopped; //1016
sigs10171024   := outRobotProgramChoice; //1017-1020
sigs10171024.4 := outRobotProgramOption1; //1021
sigs10171024.5 := outRobotProgramOption2; //1022
sigs10171024.6 := outRobotProgramOption3; //1023
sigs10171024.7 := outRobotRequestedTool.0; //1024
sigs10251032.0 := outRobotRequestedTool.1; //1025
sigs10251032.1 := outRobotRequestedTool.2; //1026
sigs10251032.2 := outRobotRequestedTool.3; //1027
sigs10251032.3 := outRobotProgramSelected; //1028
sigs10251032.4 := outRobotGoToCleanupPosition; //1029
sigs10251032.5 := outRobotMoveX; //1030
sigs10251032.6 := outRobotMoveY; //1031
sigs10251032.7 := outRobotMoveZ; //1032
sigs10331040.0 := outRobotMovePositive; //1033


inRobotMotorOn := sigs97104.0; //97
inRobotError := sigs97104.1; //98
inRobotAutomaticMode := sigs97104.2; //99
inRobotAtHome := sigs97104.3; //100
inRobotInTeach := sigs97104.4; //101
inRobotCycleStart := sigs97104.5; //102
inRobotPowerOn := sigs97104.6; //103
inRobotPoseDataIsSent := sigs97104.7; //104
inRobotEStopOn := sigs105112.0; //105
inRobotBatteryAlarm := sigs105112.1; //106
inRobotToolNumberCurrent := 0;
inRobotToolNumberCurrent := inRobotToolNumberCurrent OR (BIT_TO_USINT(sigs105112.2) * 1); //107
inRobotToolNumberCurrent := inRobotToolNumberCurrent OR (BIT_TO_USINT(sigs105112.3) * 2); //108
inRobotToolNumberCurrent := inRobotToolNumberCurrent OR (BIT_TO_USINT(sigs105112.4) * 4); //109
inRobotToolNumberCurrent := inRobotToolNumberCurrent OR (BIT_TO_USINT(sigs105112.5) * 8); //110

inRobotToolNumberRequest := 0;
inRobotToolNumberRequest := inRobotToolNumberRequest OR (BIT_TO_USINT(sigs105112.6) * 1); //111
inRobotToolNumberRequest := inRobotToolNumberRequest OR (BIT_TO_USINT(sigs105112.7) * 2); //112
inRobotToolNumberRequest := inRobotToolNumberRequest OR (BIT_TO_USINT(sigs113120.0) * 4); //113
inRobotToolNumberRequest := inRobotToolNumberRequest OR (BIT_TO_USINT(sigs113120.1) * 8); //114
inRobotReleaseTool := sigs113120.2; //115
inRobotProgramRunning := sigs113120.3; // Signal 116
inRobotToolUpdated := sigs113120.4; // Signal 117
inRobotStartofProgram := sigs113120.5; // Signal 118
// posedata.pc is running

//
END_METHOD

METHOD Update_Tool : BOOL
VAR_INPUT
	current : USINT;
	request : USINT;
END_VAR
outRobotCurrentTool := current;
outRobotRequestedTool := request;
END_METHOD

END_FUNCTION_BLOCK

// ---- POUs/Components/FB_Spindle.TcPOU
FUNCTION_BLOCK FB_Spindle
VAR_INPUT
END_VAR
VAR_OUTPUT
END_VAR
VAR
	// ================= Tool Changing ====================================
	pbToolChange AT %I*: BOOL;
	spindleToolLocked AT %I* : BOOL;
	spindleToolOpen AT %I* : BOOL;
	cylinderToolRelease1 AT %Q* : BOOL;
	cylinderToolRelease2 AT %Q* : BOOL;
	spindleClean AT %Q* : BOOL;
	toolChangeTimer : TON;
	tool0 AT %I* : BOOL;
	tool1 AT %I* : BOOL;
	tool2 AT %I* : BOOL;
	tool3 AT %I* : BOOL;
	tool4 AT %I* : BOOL;
	tool5 AT %I* : BOOL;
	tool6 AT %I* : BOOL;
	tool7 AT %I* : BOOL;
	toolLimitSwitchArray : ARRAY[0..8] OF BOOL;
	//Dust Hood
	dustHoodCylinder AT %Q*		: BOOL;
	
	currentTool : Tool_Type := GVL_Programs.noTool;
	toolSelectedAtInitialization : BOOL := FALSE;
	
	//--------------------Spindle TCP communication --------
	fbWriteRegs : FB_MBWriteRegs; //Function call
	fbWriteRegs2 : FB_MBWriteRegs; //Error reset
	fbReadReg	: FB_MBReadRegs; //Drive run/stop
	fbReadReg2	: FB_MBReadRegs; //Error
	fbReadRegSpeed	: FB_MBReadRegs; //Speed
	fbReadRegTorque	: FB_MBReadRegs; //Torque
	ipAddr      : STRING(15) := '192.168.1.5'; //IPADDRESS
	eWriteState	: (WAIT, START, STOP, WRITE); //state machine
	spindleRunStatus : WORD;
	spindleErrorStatus	: WORD;
	spindleTorqueStatus : WORD;
	spindleSpeedStatus	: WORD;
	spindleIsStopped	: BOOL;
	spindleError		: BOOL;
	spindleSpeed		: INT;
	spindleTorque		: INT;
	
	//--------------------Warmup params-----------
	spindleIsWarm 	: BOOL;
	warmupSpeed1 	: INT := 12000;
	warmupTime1 	: TIME := T#240S;
	warmupSpeed2 	: INT := 18000;
	warmupTime2 	: TIME := T#240S;
	warmupSpeed3 	: INT := 24000;
	warmupTime3 	: TIME := T#240S;
	startTime		: TIME;
	elapsedWarmupTime : TIME;
	spindleWarmupOn	: BOOL;
	triggerWarmup	: R_TRIG;
	
	warmUp3: BOOL;
	warmUp2: BOOL;
	warmUp1: BOOL;
	triggerWarm1: R_TRIG;
	triggerWarm2: R_TRIG;
	triggerWarm3: R_TRIG;
	fTrigWarm3 : F_TRIG;
	requestedTool: Tool_Type;
END_VAR

VFD_Status();
//Spindle warmup routine, trigerred from Start_Spindle and stopped with Stop_Spindle
	triggerWarmup(CLK:=spindleWarmupOn);
	triggerWarm1(CLK:=warmUp1);
	triggerWarm2(CLK:=warmUp2);
	triggerWarm3(CLK:=warmUp3);
	fTrigWarm3(CLK := warmUp3);
	
IF spindleWarmupOn THEN
	IF triggerWarmup.Q THEN
		startTime := TIME(); 
	END_IF
		
	elapsedWarmupTime := TIME() - startTime;
	
	IF elapsedWarmupTime > warmUpTime1 + warmupTime2 + warmupTime3 THEN
		warmUp1 := FALSE;
		warmUp2 := FALSE;
		warmUp3 := FALSE;
		Stop_Spindle();
		spindleWarmupOn := FALSE;
		spindleIsWarm := TRUE;
	ELSIF elapsedWarmupTime > warmUpTime1 + warmupTime2 THEN
		warmUp1 := FALSE;
		warmUp2 := FALSE;
		warmUp3 := TRUE;
	ELSIF elapsedWarmupTime > warmUpTime1 THEN
		warmUp1 := FALSE;
		warmUp2 := TRUE;
		warmUp3 := FALSE;
	ELSIF elapsedWarmupTime > T#0S THEN
		warmUp1 := TRUE;
		warmUp2 := FALSE;
		warmUp3 := FALSE;
	END_IF
	
	IF triggerWarm1.Q THEN
		Start_Spindle(spindleSpeed := warmupSpeed1);
	ELSIF triggerWarm2.Q THEN
		Start_Spindle(spindleSpeed := warmupSpeed2);
	ELSIF triggerWarm3.Q THEN
		Start_Spindle(spindleSpeed := warmupSpeed3);
	END_IF

END_IF

METHOD Dust_Hood : BOOL
VAR_INPUT
	x_pose : LREAL;
	enable : BOOL;
END_VAR
IF enable THEN
	IF x_pose < -1060 THEN
		dustHoodCylinder := FALSE;
	ELSE
		dustHoodCylinder := TRUE;
	END_IF
ELSE
	dustHoodCylinder := FALSE;
END_IF
END_METHOD

//Sets tool change cylinders to closed, returns true if tool locked
METHOD Grab_Tool : BOOL 
VAR_INPUT
END_VAR
cylinderToolRelease1 := FALSE;
cylinderToolRelease2 := FALSE;
Grab_Tool := spindleToolLocked;
END_METHOD

METHOD Manual_Tool_Change
VAR_INPUT
	changeToolEnable : BOOL;
END_VAR
IF changeToolEnable THEN
	toolChangeTimer(IN:= pbToolChange, PT:=T#2S);
	
	IF pbToolChange THEN
		IF toolChangeTimer.Q AND spindleIsStopped THEN
			cylinderToolRelease1 := TRUE;
			cylinderToolRelease2 := TRUE;
		END_IF
	ELSE
		cylinderToolRelease1 := FALSE;
		cylinderToolRelease2 := FALSE;
	END_IF
END_IF
END_METHOD

METHOD Release_Tool : BOOL; //Sets tool change cylinders to open, returns true if tool released
VAR_INPUT
END_VAR
IF spindleIsStopped THEN
	cylinderToolRelease1 := TRUE;
	cylinderToolRelease2 := TRUE;
	Release_Tool := spindleToolOpen;
ELSE
	cylinderToolRelease1 := FALSE;
	cylinderToolRelease2 := FALSE;
	Release_Tool := FALSE;
END_IF
END_METHOD

//Resets drive, returns true if no drive error
METHOD Reset_Drive : BOOL
VAR_INPUT
END_VAR
VAR
	errorReset : WORD := INT_TO_WORD(2);
END_VAR
fbWriteRegs2(
			sIPAddr:= ipAddr, 
			nTCPPort:= 502, 
			nUnitID:= 16#FF, 
			nQuantity:= 1, 
			nMBAddr:= 16#2002, 
			cbLength:= SIZEOF(errorReset), 
			pSrcAddr:= ADR(errorReset), 
			bExecute:= FALSE, 
			tTimeout:= , 
			bBusy=> , 
			bError=> , 
			nErrId=> );
			
fbWriteRegs2(
			sIPAddr:= ipAddr, 
			nTCPPort:= 502, 
			nUnitID:= 16#FF, 
			nQuantity:= 1, 
			nMBAddr:= 16#2002, 
			cbLength:= SIZEOF(errorReset), 
			pSrcAddr:= ADR(errorReset), 
			bExecute:= TRUE, 
			tTimeout:= , 
			bBusy=> , 
			bError=> , 
			nErrId=> );
			
IF NOT spindleError THEN
	Reset_Drive := TRUE;
END_IF
END_METHOD

//Starts spindle warmup, called in fbSpindle
METHOD Spindle_Warmup
VAR_INPUT
END_VAR
spindleWarmupOn := TRUE;
END_METHOD

//Description:
//This method is responsible for starting the spindle motor based on the input speed provided in revolutions per minute (RPM). It converts the spindle speed into frequency and initiates the spindle motor accordingly.

//Parameters:
//- spindleSpeed: INT - The desired spindle speed in RPM.

//Returns:
//This method does not return any value.
METHOD Start_Spindle
VAR_INPUT
	spindleSpeed : INT; //Spindle speed RPM
	
END_VAR

VAR
	spindleFrequency : INT := (spindleSpeed - 12000) / 30 + 400; //Speed conversion to frequency
	startValue  : ARRAY [0..1] OF WORD := [INT_TO_WORD(18), INT_TO_WORD(SpindleFrequency*10)];
END_VAR
fbWriteRegs(
			sIPAddr:= ipAddr, 
			nTCPPort:= 502, 
			nUnitID:= 16#FF, 
			nQuantity:= 2, 
			nMBAddr:= 16#2000, 
			cbLength:= SIZEOF(startValue), 
			pSrcAddr:= ADR(startValue), 
			bExecute:= FALSE, 
			tTimeout:= , 
			bBusy=> , 
			bError=> , 
			nErrId=> );
			
fbWriteRegs(
			sIPAddr:= ipAddr, 
			nTCPPort:= 502, 
			nUnitID:= 16#FF, 
			nQuantity:= 2, 
			nMBAddr:= 16#2000, 
			cbLength:= SIZEOF(startValue), 
			pSrcAddr:= ADR(startValue), 
			bExecute:= TRUE, 
			tTimeout:= , 
			bBusy=> , 
			bError=> , 
			nErrId=> );
			
spindleClean := TRUE;
END_METHOD

//Stops spindle
METHOD Stop_Spindle
VAR_INPUT
END_VAR

VAR
	stopValue: ARRAY [0..1] OF WORD := [INT_TO_WORD(1), INT_TO_WORD(0)];
END_VAR
fbWriteRegs(
			sIPAddr:= ipAddr, 
			nTCPPort:= 502, 
			nUnitID:= 16#FF, 
			nQuantity:= 2, 
			nMBAddr:= 16#2000, 
			cbLength:= SIZEOF(stopValue), 
			pSrcAddr:= ADR(stopValue), 
			bExecute:= FALSE, 
			tTimeout:= , 
			bBusy=> , 
			bError=> , 
			nErrId=> );

fbWriteRegs(
			sIPAddr:= ipAddr, 
			nTCPPort:= 502, 
			nUnitID:= 16#FF, 
			nQuantity:= 2, 
			nMBAddr:= 16#2000, 
			cbLength:= SIZEOF(stopValue), 
			pSrcAddr:= ADR(stopValue), 
			bExecute:= TRUE, 
			tTimeout:= , 
			bBusy=> , 
			bError=> , 
			nErrId=> );
			
spindleWarmupOn := FALSE;
warmup1 := FALSE;
warmup2 := FALSE;
warmup3 := FALSE;
spindleClean := FALSE;
END_METHOD

//Updates the current tool based on an integer
METHOD Update_Current_Tool : BOOL
VAR_INPUT
	toolNumber : INT;
END_VAR
VAR
	updatedTool : Tool_Type;
	success : BOOL;
END_VAR
success := TRUE;
CASE toolNumber OF
		0:
			updatedTool := GVL_Programs.sawblade;
		6:
			updatedTool := GVL_Programs.halfInchBall;
		2:
			updatedTool := GVL_Programs.quarterInchUpcut;
		5:
			updatedTool := GVL_Programs.dovetail;
		4:
			updatedTool := GVL_Programs.halfInchUpcut;
		8:
			updatedTool := GVL_Programs.noTool;
			
		ELSE
			success := FALSE;
	END_CASE
		
currentTool := updatedTool;
	
// Successfully updated the current tool
IF NOT success THEN
	Update_Current_Tool := FALSE;
ELSE
	Update_Current_Tool := TRUE;
	toolSelectedAtInitialization := TRUE;
END_IF
END_METHOD

METHOD Update_Requested_Tool : BOOL
VAR_INPUT
	toolNumber : INT;
END_VAR
VAR
	updatedTool : Tool_Type;
	success : BOOL;
END_VAR
CASE toolNumber OF
		0:
			updatedTool := GVL_Programs.sawblade;
		6:
			updatedTool := GVL_Programs.halfInchBall;
		2:
			updatedTool := GVL_Programs.quarterInchUpcut;
		5:
			updatedTool := GVL_Programs.dovetail;
		4:
			updatedTool := GVL_Programs.halfInchUpcut;
		8:
			updatedTool := GVL_Programs.noTool;
			
		ELSE
			success := FALSE;
	END_CASE
		
requestedTool := updatedTool;
	
// Successfully updated the current tool
IF NOT success THEN
	Update_Requested_Tool := FALSE;
ELSE
	Update_Requested_Tool := TRUE;
END_IF
END_METHOD

METHOD Verify_Tool_Change_Request : BOOL
VAR_INPUT
	toolToDrop : UINT;
	toolToPickup : UINT;
END_VAR
//NC contacts. Detect if current tool holder is empty and requested tool holder is full. If no tool is selected, checks if spindle is empty
toolLimitSwitchArray[0] := tool0;
toolLimitSwitchArray[1] := tool1;
toolLimitSwitchArray[2] := tool2;
toolLimitSwitchArray[3] := tool3;
toolLimitSwitchArray[4] := tool4;
toolLimitSwitchArray[5] := tool5;
toolLimitSwitchArray[6] := tool6;
toolLimitSwitchArray[7] := tool7;

IF (toolLimitSwitchArray[toolToDrop] OR toolToDrop = 8) AND (NOT toolLimitSwitchArray[toolToPickup] OR toolToPickup = 8) OR (toolToDrop = toolToPickup AND toolLimitSwitchArray[toolToDrop]) THEN 
	Verify_Tool_Change_Request := TRUE;
ELSE
	Verify_Tool_Change_Request := FALSE;
END_IF
//Verify_Tool_Change_Request := TRUE; //TODO: remove once wired!!
END_METHOD

//Updates the status of the VFD: whether it's stopped and whether it is in error state
METHOD VFD_Status : BOOL //returns true if drive has no error
VAR_INPUT
END_VAR
VAR
	runStatus : USINT;
	errorStatus : USINT;
END_VAR
fbReadReg(
			sIPAddr:= ipAddr, 
			nTCPPort:= 502, 
			nUnitID:= 16#FF, 
			nQuantity:= 1, 
			nMBAddr:= 16#2101, 
			cbLength:= SIZEOF(spindleRunStatus), 
			pDestAddr := ADR(spindleRunStatus), 
			bExecute:= FALSE, 
			tTimeout:= , 
			bBusy=> , 
			bError=> , 
			nErrId=> );
			
fbReadReg(
			sIPAddr:= ipAddr, 
			nTCPPort:= 502, 
			nUnitID:= 16#FF, 
			nQuantity:= 1, 
			nMBAddr:= 16#2101, 
			cbLength:= SIZEOF(spindleRunStatus), 
			pDestAddr := ADR(spindleRunStatus), 
			bExecute:= TRUE, 
			tTimeout:= , 
			bBusy=> , 
			bError=> , 
			nErrId=> );
			
fbReadReg2(
			sIPAddr:= ipAddr, 
			nTCPPort:= 502, 
			nUnitID:= 16#FF, 
			nQuantity:= 1, 
			nMBAddr:= 16#2226, 
			cbLength:= SIZEOF(spindleErrorStatus), 
			pDestAddr := ADR(spindleErrorStatus), 
			bExecute:= FALSE, 
			tTimeout:= , 
			bBusy=> , 
			bError=> , 
			nErrId=> );

fbReadReg2(
			sIPAddr:= ipAddr, 
			nTCPPort:= 502, 
			nUnitID:= 16#FF, 
			nQuantity:= 1, 
			nMBAddr:= 16#2226, 
			cbLength:= SIZEOF(spindleErrorStatus), 
			pDestAddr := ADR(spindleErrorStatus), 
			bExecute:= TRUE, 
			tTimeout:= , 
			bBusy=> , 
			bError=> , 
			nErrId=> );
			
fbReadRegSpeed(
			sIPAddr:= ipAddr, 
			nTCPPort:= 502, 
			nUnitID:= 16#FF, 
			nQuantity:= 1, 
			nMBAddr:= 16#210C, 
			cbLength:= SIZEOF(spindleSpeedStatus), 
			pDestAddr := ADR(spindleSpeedStatus), 
			bExecute:= FALSE, 
			tTimeout:= , 
			bBusy=> , 
			bError=> , 
			nErrId=> );

fbReadRegSpeed(
			sIPAddr:= ipAddr, 
			nTCPPort:= 502, 
			nUnitID:= 16#FF, 
			nQuantity:= 1, 
			nMBAddr:= 16#210C, 
			cbLength:= SIZEOF(spindleSpeedStatus), 
			pDestAddr := ADR(spindleSpeedStatus), 
			bExecute:= TRUE, 
			tTimeout:= , 
			bBusy=> , 
			bError=> , 
			nErrId=> );
			
fbReadRegTorque(
			sIPAddr:= ipAddr, 
			nTCPPort:= 502, 
			nUnitID:= 16#FF, 
			nQuantity:= 1, 
			nMBAddr:= 16#210B, 
			cbLength:= SIZEOF(spindleTorqueStatus), 
			pDestAddr := ADR(spindleTorqueStatus), 
			bExecute:= FALSE, 
			tTimeout:= , 
			bBusy=> , 
			bError=> , 
			nErrId=> );
fbReadRegTorque(
			sIPAddr:= ipAddr, 
			nTCPPort:= 502, 
			nUnitID:= 16#FF, 
			nQuantity:= 1, 
			nMBAddr:= 16#210B, 
			cbLength:= SIZEOF(spindleTorqueStatus), 
			pDestAddr := ADR(spindleTorqueStatus), 
			bExecute:= TRUE, 
			tTimeout:= , 
			bBusy=> , 
			bError=> , 
			nErrId=> );

runStatus := WORD_TO_USINT(spindleRunStatus);
IF runStatus.0 = 0 AND runStatus.1 = 0 THEN
	spindleIsStopped := TRUE;
ELSE 
	spindleIsStopped := FALSE;
END_IF

errorStatus := WORD_TO_USINT(spindleErrorStatus);
IF errorStatus.3 = 1 AND errorStatus.2 = 0 THEN
	spindleError := TRUE;
ELSE 
	spindleError := FALSE;
END_IF

spindleSpeed := WORD_TO_INT(SpindleSpeedStatus);
spindleTorque := WORD_TO_INT(SpindleTorqueStatus);

VFD_Status := NOT spindleError;
END_METHOD

END_FUNCTION_BLOCK

// ---- POUs/Components/FB_GantryHoldDown.TcPOU
//TODO: set methods to enable all following, pneumatic cylinder activation, error handling

FUNCTION_BLOCK FB_GantryHoldDown
VAR_OUTPUT
END_VAR
VAR
	//MC_functions, called in methods
	fbMC_PowerWest		: MC_Power;
	fbMC_PowerEast		: MC_Power;
	fbMC_HomeWest		: MC_Home;
	fbMC_HomeEast		: MC_Home;
	fbMC_MoveAbsWest1	: MC_MoveAbsolute;
	fbMC_MoveAbsWest2	: MC_MoveAbsolute;
	fbMC_MoveVelocity: MC_MoveVelocity;
	fbMC_SyncAxes		: MC_GearIn;
	fbReadStatus		: MC_ReadStatus;
	fbMC_Stop			: MC_Stop;
	fbMC_Halt			: MC_HALT;
	Aborting			: MC_BufferMode;
	fbMC_Reset			: MC_Reset;
	fbSOEReset			: FB_SoEReset;
	
	//Inputs
	ls1NE AT %I* 		: BOOL;
	ls3NW AT %I* 		: BOOL;
	
	//Pneumatic cylinders
	cylindersNorth 			AT %Q* : BOOL;
	cylindersCentreNorth	AT %Q* : BOOL;
	cylindersCentreSouth	AT %Q* : BOOL;
	cylindersSouth			AT %Q* : BOOL;
	pressureSwitchSpindle	AT %I* : BOOL;
	pressureSwitchHoldDown	AT %I* : BOOL;
	pressureSwitchTableClamps AT %I* : BOOL;
	pressureSwitchTimer : TON;
	
	//Pneumatic switches
	
	rollersReady		: BOOL;
	
	// Enable bools
	executeEnable		: BOOL := FALSE;
	executeHome 		: BOOL := FALSE;
	executeCouple 		: BOOL := FALSE;
	executeCylinders	: BOOL := FALSE;
	followVariable		: BOOL:= TRUE; //Set for following robot
	stopGantry			: BOOL := FALSE;
	resetExec			: BOOL := FALSE;
	executeManualMove		: BOOL;
	executeHalt			: BOOL;
	manualMoveDirection 		: MC_Direction;
END_VAR

GVL_Axes.AxisWest.ReadStatus();
GVL_Axes.AxisEast.ReadStatus();
	
// Movement functions
Servo_Commands();
// Enable and couple axes
executeEnable := TRUE;
IF GVL_Axes.AxisEast.NcToPlc.CoupleState <> 3 THEN
	executeCouple := NOT executeCouple;
END_IF

METHOD Cylinder_Set_Cutting
VAR_INPUT
END_VAR
VAR
	POS_CYLINDER_NORTH : LREAL := 76.5; //mm, position of north pneum cylinder relative to gantry plate
	POS_CYLINDER_NORTHCENTRE : LREAL := 229.62; //mm, position of centre north pneum cylinder relative to gantry plate
	POS_CYLINDER_SOUTHCENTRE : LREAL := 712.212; //mm, position of centre south pneum cylinder relative to gantry plate
	POS_CYLINDER_SOUTH : LREAL := 867.832; //mm, position of south pneum cylinder relative to gantry plate
	POS_TABLE_NORTH : LREAL := 474.14; //mm, position of table start WRT Zero
	FACTOR_OF_SAFETY : LREAL := 100; //mm, distance from edge of table cylinders will rise
END_VAR
IF GVL_Axes.AxisWest.NcToPlc.ActPos < POS_TABLE_NORTH + FACTOR_OF_SAFETY - POS_CYLINDER_NORTH THEN
	cylindersNorth := 1;
ELSE
	cylindersNorth := 0;
END_IF

IF GVL_Axes.AxisWest.NcToPlc.ActPos < POS_TABLE_NORTH + FACTOR_OF_SAFETY - POS_CYLINDER_NORTHCENTRE THEN
	cylindersCentreNorth := 1;
ELSE
	cylindersCentreNorth := 0;
END_IF

IF GVL_Axes.AxisWest.NcToPlc.ActPos > POS_TABLE_NORTH + GVL_SERVO_ROBOT_CONST.LEN_WOOD - FACTOR_OF_SAFETY - POS_CYLINDER_SOUTH THEN
	cylindersSouth := 1;
ELSE
	cylindersSouth := 0;
END_IF

IF GVL_Axes.AxisWest.NcToPlc.ActPos > POS_TABLE_NORTH + GVL_SERVO_ROBOT_CONST.LEN_WOOD - FACTOR_OF_SAFETY - POS_CYLINDER_SOUTHCENTRE THEN
		cylindersCentreSouth := 1;
ELSE 
		cylindersCentreSouth := 0;
END_IF
END_METHOD

METHOD Follow_Robot : BOOL //returns false if robot too far away (1"), true if it is
VAR_INPUT
	robotPoseGantry : Structure_RobotPose;
END_VAR

VAR
	targetPosition: LREAL;
	accel: LREAL:=600;
	decel: LREAL:=600;
	jer:   LREAL:=1200;
	vel: LREAL:= 170;
	
	dustBootBottom : INT := 20;
	dustBootLeft : INT := 20;
	dustBootRight : INT := 20;
	dustBootTop : INT := 20;
END_VAR
//Set target position to middle of robot tool
targetPosition := (robotPoseGantry.yPose - GVL_SERVO_ROBOT_CONST.MIN_POS_ROBOT) * GVL_SERVO_ROBOT_CONST.DIFFERENCE_SERVOWEST/GVL_SERVO_ROBOT_CONST.DIFFERENCE_ROBOT;

//If target position - current position > threshold, hold robot
IF ABS(targetPosition - GVL_Axes.AxisWest.NcToPlc.ActPos) > GVL_SERVO_ROBOT_CONST.FOLLOW_THRESHOLD
AND (robotPoseGantry.zPose < GVL_SERVO_ROBOT_CONST.ROLLERS_Z_HEIGHT) THEN
//OR ((cylindersCentreNorth OR cylindersNorth) AND NOT GVL_Axes.AxisWest.Status.PositiveDirection)
//OR ((cylindersCentreSouth OR cylindersSouth) AND NOT GVL_Axes.AxisWest.Status.NegativeDirection)) THEN
		Follow_Robot := FALSE; //Gantry isn't following, hold robot
ELSE 
	Follow_Robot := TRUE; //Gantry is following properly, keep robot on run
END_IF

IF targetPosition < GVL_SERVO_ROBOT_CONST.MIN_POS_SERVOWEST THEN
	targetPosition := GVL_SERVO_ROBOT_CONST.MIN_POS_SERVOWEST;
ELSIF targetPosition > GVL_SERVO_ROBOT_CONST.MAX_POS_SERVOWEST THEN
	targetPosition := GVL_SERVO_ROBOT_CONST.MAX_POS_SERVOWEST;
END_IF

followVariable := NOT followVariable;

IF GVL_Axes.AxisWest.Status.Homed THEN
	fbMC_MoveAbsWest1(
		Axis:= GVL_Axes.AxisWest, 
		Execute:= followVariable, 
		Position:= targetPosition, 
		Velocity:= vel,
		Acceleration:= accel, 
		Deceleration:= decel,
		Jerk:= jer, 
		BufferMode:= Aborting);
	
	fbMC_MoveAbsWest2(
		Axis:= GVL_Axes.AxisWest, 
		Execute:= NOT followVariable, 
		Position:= targetPosition, 
		Velocity:= vel,
		Acceleration:= accel, 
		Deceleration:= decel,
		Jerk:= jer, 
		BufferMode:= Aborting);
END_IF
END_METHOD

//Enables, couples and homes hold down gantry
//TODO: check if robot is above rollers before homing
//Returns True if can sucessfully home, false if robot too low
METHOD Home_Servos : Structure_Error
VAR_INPUT
	robotPose	: Structure_RobotPose;
END_VAR

VAR

END_VAR
IF robotPose.zPose > GVL_SERVO_ROBOT_CONST.ROLLERS_Z_HEIGHT THEN
	//Home Axes
	IF GVL_Axes.AxisEast.NcToPlc.CoupleState = 3 THEN
		executeHome := TRUE;
		Home_Servos.isError := FALSE;
		Home_Servos.errorMessage := 'No Error';
	ELSE
		Home_Servos.isError := TRUE;
		Home_Servos.errorMessage := 'Axis not coupled properly';
	END_IF
ELSE
	Home_Servos.isError := TRUE;
	Home_Servos.errorMessage := 'Robot too low to home';
END_IF
END_METHOD

METHOD Lower_Raise_Rollers
VAR_INPUT
	raiseRollers	: BOOL;
END_VAR
cylindersNorth 			:= raiseRollers;
cylindersCentreNorth	:= raiseRollers;
cylindersCentreSouth 	:= raiseRollers;
cylindersSouth 			:= raiseRollers;
END_METHOD

METHOD Manual_Move_Servos : BOOL
VAR_INPUT
	direction : INT; //1 for south, -1 for north
	moveServos : BOOL; //True to move
END_VAR
IF moveServos THEN
	IF direction = -1 THEN
		manualMoveDirection := MC_Negative_Direction;
	ELSE
		manualMoveDirection := MC_Positive_Direction;
	END_IF
	
	executeHalt := FALSE;
	executeManualMove := TRUE;
ELSE
	executeHalt := TRUE;
	executeManualMove := FALSE;
END_IF
END_METHOD

METHOD Pneumatics_Error : Structure_Error
VAR_INPUT
END_VAR
Pneumatics_Error.errorMessage := '';

IF NOT (pressureSwitchSpindle AND  pressureSwitchHoldDown AND pressureSwitchTableClamps) THEN
	pressureSwitchTimer(IN:= TRUE, PT:=T#5S);
ELSE
	pressureSwitchTimer(IN:= FALSE, PT:=T#5S);
END_IF


IF NOT pressureSwitchTimer.Q THEN
	Pneumatics_Error.isError := FALSE;
ELSE
	Pneumatics_Error.isError := TRUE;
	IF NOT pressureSwitchSpindle THEN
		Pneumatics_Error.errorMessage := CONCAT(Pneumatics_Error.errorMessage, '\nPressure Switch Spindle Off');
	END_IF
	IF NOT pressureSwitchHoldDown THEN
		Pneumatics_Error.errorMessage := CONCAT(Pneumatics_Error.errorMessage, '\nPressure Switch HoldDown Off');
	END_IF
	IF NOT pressureSwitchTableClamps THEN
		Pneumatics_Error.errorMessage := CONCAT(Pneumatics_Error.errorMessage, '\nPressure Switch Table Clamps Off');
	END_IF
END_IF
END_METHOD

//Resets servo errors
METHOD Reset_Servos : BOOL // Returns true if errors reset successfully
VAR_INPUT
END_VAR
stopGantry := FALSE;
resetExec := TRUE;

Reset_Servos := NOT GVL_Axes.AxisWest.Status.Error;
IF Reset_Servos THEN
	resetExec := FALSE;
END_IF
END_METHOD

//All the servo motions. Triggered in separate methods by their execute flags
METHOD Servo_Commands
VAR_INPUT
END_VAR

VAR
	Execute: BOOL;
END_VAR
//Enable Axes
fbMC_PowerWest(
	Axis:= GVL_Axes.AxisWest, 
	Enable:= executeEnable, 
	Enable_Positive:= executeEnable, 
	Enable_Negative:= executeEnable, 
	Override:= 100.0);
		
fbMC_PowerEast(
	Axis:= GVL_Axes.AxisEast, 
	Enable:= executeEnable, 
	Enable_Positive:= executeEnable, 
	Enable_Negative:= executeEnable, 
	Override:= 100.0);
	
//Couple Axes
fbMC_SyncAxes(
	Master:= GVL_Axes.AxisWest, 
	Slave:= GVL_Axes.AxisEast, 
	Execute:= executeCouple, 
	RatioNumerator:= 1);

//Home
fbMC_HomeWest(
	Axis:= GVL_Axes.AxisWest, 
	Execute:= executeHome, 
	Position:= GVL_SERVO_ROBOT_CONST.POSITION_LIMIT_SWITCH, 
	HomingMode:= MC_DefaultHoming, 
	bCalibrationCam:= NOT ls3NW);
	
IF fbMC_HomeWest.Done THEN
	executeHome := FALSE;
END_IF

fbMC_MoveVelocity(
	Axis := GVL_Axes.AxisWest, 
   	Execute := executeManualMove, 
	Velocity := 50,
Direction :=  manualMoveDirection);

fbMC_Halt(
	Axis := GVL_Axes.AxisWest,
	Execute := executeHalt);
	
//Stop
fbMC_Stop(
	Axis:= GVL_Axes.AxisWest, 
	Execute:= stopGantry, 
	);
	
//Reset
fbMC_Reset(
	Axis := GVL_Axes.AxisWest,
	Execute := ResetExec);
	
	fbMC_Reset(
	Axis := GVL_Axes.AxisEast,
	Execute := ResetExec);
END_METHOD

//Stops gantry
METHOD Stop_Servos : BOOL
VAR_INPUT
END_VAR
stopGantry := TRUE;
END_METHOD

END_FUNCTION_BLOCK

// ---- POUs/Components/FB_Enclosure.TcPOU
FUNCTION_BLOCK FB_Enclosure
VAR
	// =============== Table clamping  ================================================
	pbTableWest				AT %I* : BOOL;
	pbTableEast				AT %I* : BOOL;

	pbTableWestLast: BOOL;
	pbTableEastLast: BOOL;
	cylinderTableWest		AT %Q* : BOOL := FALSE;
	cylinderTableEast		AT %Q* : BOOL := FALSE;
	
	// Door
	openCloseDoor				AT %Q* : BOOL;
	enableRollingDoor 			AT %Q* : BOOL := TRUE;
	doorIsClosed				AT %I* : BOOL;
	doorTimer				: TON;
	startTimer: BOOL;
	
	dustCollectionOn : BOOL;
END_VAR

// Reverts door to pushbutton operation once 0.5s has passed
IF startTimer THEN
	doorTimer(IN:=TRUE, PT:=T#500MS);
END_IF

IF doorTimer.Q THEN
	openCloseDoor := FALSE;
	doorTimer(IN:=FALSE);
	startTimer := FALSE;
END_IF

//Opens and closes door
METHOD Rolling_Door_HMI_Operation
VAR_INPUT
END_VAR
openCloseDoor := TRUE;
startTimer := TRUE;
END_METHOD

METHOD Table_Clamp_Control_HMI
VAR_INPUT
	eastTableLock : BOOL;
	westTableLock : BOOL;
END_VAR
cylinderTableWest := westTableLock;
cylinderTableEast := eastTableLock;
END_METHOD

METHOD Table_Clamp_Control_Pushbutton : BOOL
VAR_INPUT
END_VAR
IF pbTableWest AND NOT pbTableWestLast THEN
	cylinderTableWest := NOT cylinderTableWest;
END_IF

pbTableWestLast := pbTableWest;

IF pbTableEast AND NOT pbTableEastLast THEN
	cylinderTableEast := NOT cylinderTableEast;
END_IF

pbTableEastLast := pbTableEast;
END_METHOD

END_FUNCTION_BLOCK

// ---- POUs/Components/FB_TorqueSensor.TcPOU
FUNCTION_BLOCK FB_TorqueSensor
VAR_INPUT
END_VAR
VAR_OUTPUT
END_VAR
VAR
	countsPerForce : LREAL := 80000;
	countsPerTorque : LREAL := 1000000;
	FxCounts AT %I* : DINT;
	FyCounts AT %I* : DINT;
	FzCounts AT %I* : DINT;
	TxCounts AT %I* : DINT;
	TyCounts AT %I* : DINT;
	TzCounts AT %I* : DINT;
	xForce	: LREAL;
	yForce : LREAL;
	zForce : LREAL;
	xTorque : LREAL;
	yTorque : LREAL;
	zTorque : LREAL;
END_VAR

xForce := FxCounts / countsPerForce;
yForce := FyCounts / countsPerForce;
zForce := FzCounts / countsPerForce;
xTorque := TxCounts / countsPerTorque;
yTorque := TyCounts / countsPerTorque;
zTorque := TzCounts / countsPerTorque;

END_FUNCTION_BLOCK

// ---- POUs/Components/FB_OperatingCounter.TcPOU
FUNCTION_BLOCK FB_OperatingCounter
VAR_INPUT
	stateString : STRING;
END_VAR
VAR_OUTPUT
END_VAR
VAR
	// Timer to count operating time
    runTimer : TON; // Timer On-Delay
    elapsedTime : TIME := T#0S; // Time elapsed since last increment

    // Time interval for incrementing operating hours (e.g., every second)
    timeInterval : TIME := T#1S;

    totalRunHoursRounded : INT;
END_VAR

totalRunHoursRounded := REAL_TO_INT(GVL_OperationCounter.totalRunHours);

IF stateString = 'RUN' OR stateString = 'TOOLCHANGERUN' OR stateString = 'TOOLCHANGEINIT' THEN
	// Timer setup
	runTimer(IN := TRUE, PT := timeInterval);
	elapsedTime := runTimer.ET;
	
	// Check if the timer has elapsed
	IF runTimer.Q THEN
		// Increment operating hours (timeInterval is in seconds, convert to hours)
		GVL_OperationCounter.totalRunHours := GVL_OperationCounter.totalRunHours + TIME_TO_REAL(elapsedTime) / 3600000.0;
		// Reset timer
		runTimer(IN := FALSE);
		runTimer(IN := TRUE);
	END_IF
END_IF

END_FUNCTION_BLOCK
